	X =  480.566  mm,	Y =   -445.856  mm,	Z =   -229.363  mm,
	W =  90.000 deg,	P =   0.000 deg,	R =   90.000 deg
};
P[2287]{
   GP1:
	UF : 0, UT : 6,		CONFIG : 'N U T, 0, 0, 0',
	X =  481.182  mm,	Y =   -445.586  mm,	Z =   -229.154  mm,
	W =  90.000 deg,	P =   0.000 deg,	R =   90.000 deg
};
P[2288]{
   GP1:
	UF : 0, UT : 6,		CONFIG : 'N U T, 0, 0, 0',
	X =  482.170  mm,	Y =   -444.919  mm,	Z =   -229.387  mm,
	W =  90.000 deg,	P =   0.000 deg,	R =   90.000 deg
};
P[2289]{
   GP1:
	UF : 0, UT : 6,		CONFIG : 'N U T, 0, 0, 0',
	X =  483.233  mm,	Y =   -444.478  mm,	Z =   -228.968  mm,
	W =  90.000 deg,	P =   0.000 deg,	R =   90.000 deg
};
P[2290]{
   GP1:
	UF : 0, UT : 6,		CONFIG : 'N U T, 0, 0, 0',
	X =  484.850  mm,	Y =   -443.422  mm,	Z =   -229.266  mm,
	W =  90.000 deg,	P =   0.000 deg,	R =   90.000 deg
};
P[2291]{
   GP1:
	UF : 0, UT : 6,		CONFIG : 'N U T, 0, 0, 0',
	X =  485.668  mm,	Y =   -442.930  mm,	Z =   -229.313  mm,
	W =  90.000 deg,	P =   0.000 deg,	R =   90.000 deg
};
P[2292]{
   GP1:
	UF : 0, UT : 6,		CONFIG : 'N U T, 0, 0, 0',
	X =  487.431  mm,	Y =   -441.948  mm,	Z =   -229.227  mm,
	W =  90.000 deg,	P =   0.000 deg,	R =   90.000 deg
};
P[2293]{
   GP1:
	UF : 0, UT : 6,		CONFIG : 'N U T, 0, 0, 0',
	X =  488.798  mm,	Y =   -441.282  mm,	Z =   -228.926  mm,
	W =  90.000 deg,	P =   0.000 deg,	R =   90.000 deg
};
P[2294]{
   GP1:
	UF : 0, UT : 6,		CONFIG : 'N U T, 0, 0, 0',
	X =  492.018  mm,	Y =   -439.329  mm,	Z =   -229.155  mm,
	W =  90.000 deg,	P =   0.000 deg,	R =   90.000 deg
};
P[2295]{
   GP1:
	UF : 0, UT : 6,		CONFIG : 'N U T, 0, 0, 0',
	X =  493.252  mm,	Y =   -438.538  mm,	Z =   -229.345  mm,
	W =  90.000 deg,	P =   0.000 deg,	R =   90.000 deg
};
P[2296]{
   GP1:
	UF : 0, UT : 6,		CONFIG : 'N U T, 0, 0, 0',
	X =  494.374  mm,	Y =   -438.005  mm,	Z =   -229.066  mm,
	W =  90.000 deg,	P =   0.000 deg,	R =   90.000 deg
};
P[2297]{
   GP1:
	UF : 0, UT : 6,		CONFIG : 'N U T, 0, 0, 0',
	X =  495.502  mm,	Y =   -437.305  mm,	Z =   -229.186  mm,
	W =  90.000 deg,	P =   0.000 deg,	R =   90.000 deg
};
P[2298]{
   GP1:
	UF : 0, UT : 6,		CONFIG : 'N U T, 0, 0, 0',
	X =  496.386  mm,	Y =   -436.731  mm,	Z =   -229.340  mm,
	W =  90.000 deg,	P =   0.000 deg,	R =   90.000 deg
};
P[2299]{
   GP1:
	UF : 0, UT : 6,		CONFIG : 'N U T, 0, 0, 0',
	X =  497.271  mm,	Y =   -436.217  mm,	Z =   -229.347  mm,
	W =  90.000 deg,	P =   0.000 deg,	R =   90.000 deg
};
P[2300]{
   GP1:
	UF : 0, UT : 6,		CONFIG : 'N U T, 0, 0, 0',
	X =  498.310  mm,	Y =   -435.633  mm,	Z =   -229.309  mm,
	W =  90.000 deg,	P =   0.000 deg,	R =   90.000 deg
};
P[2301]{
   GP1:
	UF : 0, UT : 6,		CONFIG : 'N U T, 0, 0, 0',
	X =  499.714  mm,	Y =   -434.837  mm,	Z =   -229.273  mm,
	W =  90.000 deg,	P =   0.000 deg,	R =   90.000 deg
};
P[2302]{
   GP1:
	UF : 0, UT : 6,		CONFIG : 'N U T, 0, 0, 0',
	X =  500.828  mm,	Y =   -434.198  mm,	Z =   -229.203  mm,
	W =  90.000 deg,	P =   0.000 deg,	R =   90.000 deg
};
P[2303]{
   GP1:
	UF : 0, UT : 6,		CONFIG : 'N U T, 0, 0, 0',
	X =  502.097  mm,	Y =   -433.246  mm,	Z =   -229.316  mm,
	W =  90.000 deg,	P =   0.000 deg,	R =   90.000 deg
};
P[2304]{
   GP1:
	UF : 0, UT : 6,		CONFIG : 'N U T, 0, 0, 0',
	X =  503.730  mm,	Y =   -431.797  mm,	Z =   -229.261  mm,
	W =  90.000 deg,	P =   0.000 deg,	R =   90.000 deg
};
P[2305]{
   GP1:
	UF : 0, UT : 6,		CONFIG : 'N U T, 0, 0, 0',
	X =  504.332  mm,	Y =   -431.117  mm,	Z =   -229.304  mm,
	W =  90.000 deg,	P =   0.000 deg,	R =   90.000 deg
};
P[2306]{
   GP1:
	UF : 0, UT : 6,		CONFIG : 'N U T, 0, 0, 0',
	X =  505.528  mm,	Y =   -429.350  mm,	Z =   -229.315  mm,
	W =  90.000 deg,	P =   0.000 deg,	R =   90.000 deg
};
P[2307]{
   GP1:
	UF : 0, UT : 6,		CONFIG : 'N U T, 0, 0, 0',
	X =  506.145  mm,	Y =   -428.643  mm,	Z =   -228.908  mm,
	W =  90.000 deg,	P =   0.000 deg,	R =   90.000 deg
};
P[2308]{
   GP1:
	UF : 0, UT : 6,		CONFIG : 'N U T, 0, 0, 0',
	X =  506.322  mm,	Y =   -427.681  mm,	Z =   -229.271  mm,
	W =  90.000 deg,	P =   0.000 deg,	R =   90.000 deg
};
P[2309]{
   GP1:
	UF : 0, UT : 6,		CONFIG : 'N U T, 0, 0, 0',
	X =  506.669  mm,	Y =   -427.189  mm,	Z =   -228.972  mm,
	W =  90.000 deg,	P =   0.000 deg,	R =   90.000 deg
};
P[2310]{
   GP1:
	UF : 0, UT : 6,		CONFIG : 'N U T, 0, 0, 0',
	X =  507.163  mm,	Y =   -425.222  mm,	Z =   -228.904  mm,
	W =  90.000 deg,	P =   0.000 deg,	R =   90.000 deg
};
P[2311]{
   GP1:
	UF : 0, UT : 6,		CONFIG : 'N U T, 0, 0, 0',
	X =  507.195  mm,	Y =   -423.814  mm,	Z =   -229.152  mm,
	W =  90.000 deg,	P =   0.000 deg,	R =   90.000 deg
};
P[2312]{
   GP1:
	UF : 0, UT : 6,		CONFIG : 'N U T, 0, 0, 0',
	X =  506.821  mm,	Y =   -419.984  mm,	Z =   -228.966  mm,
	W =  90.000 deg,	P =   0.000 deg,	R =   90.000 deg
};
P[2313]{
   GP1:
	UF : 0, UT : 6,		CONFIG : 'N U T, 0, 0, 0',
	X =  506.580  mm,	Y =   -419.034  mm,	Z =   -228.929  mm,
	W =  90.000 deg,	P =   0.000 deg,	R =   90.000 deg
};
P[2314]{
   GP1:
	UF : 0, UT : 6,		CONFIG : 'N U T, 0, 0, 0',
	X =  506.090  mm,	Y =   -418.254  mm,	Z =   -229.258  mm,
	W =  90.000 deg,	P =   0.000 deg,	R =   90.000 deg
};
P[2315]{
   GP1:
	UF : 0, UT : 6,		CONFIG : 'N U T, 0, 0, 0',
	X =  505.684  mm,	Y =   -417.150  mm,	Z =   -229.023  mm,
	W =  90.000 deg,	P =   0.000 deg,	R =   90.000 deg
};
P[2316]{
   GP1:
	UF : 0, UT : 6,		CONFIG : 'N U T, 0, 0, 0',
	X =  505.249  mm,	Y =   -416.523  mm,	Z =   -229.335  mm,
	W =  90.000 deg,	P =   0.000 deg,	R =   90.000 deg
};
P[2317]{
   GP1:
	UF : 0, UT : 6,		CONFIG : 'N U T, 0, 0, 0',
	X =  504.966  mm,	Y =   -415.874  mm,	Z =   -229.110  mm,
	W =  90.000 deg,	P =   0.000 deg,	R =   90.000 deg
};
P[2318]{
   GP1:
	UF : 0, UT : 6,		CONFIG : 'N U T, 0, 0, 0',
	X =  504.322  mm,	Y =   -414.678  mm,	Z =   -228.999  mm,
	W =  90.000 deg,	P =   0.000 deg,	R =   90.000 deg
};
P[2319]{
   GP1:
	UF : 0, UT : 6,		CONFIG : 'N U T, 0, 0, 0',
	X =  501.872  mm,	Y =   -410.680  mm,	Z =   -229.341  mm,
	W =  90.000 deg,	P =   0.000 deg,	R =   90.000 deg
};
P[2320]{
   GP1:
	UF : 0, UT : 6,		CONFIG : 'N U T, 0, 0, 0',
	X =  501.465  mm,	Y =   -409.684  mm,	Z =   -228.933  mm,
	W =  90.000 deg,	P =   0.000 deg,	R =   90.000 deg
};
P[2321]{
   GP1:
	UF : 0, UT : 6,		CONFIG : 'N U T, 0, 0, 0',
	X =  500.200  mm,	Y =   -407.765  mm,	Z =   -229.313  mm,
	W =  90.000 deg,	P =   0.000 deg,	R =   90.000 deg
};
P[2322]{
   GP1:
	UF : 0, UT : 6,		CONFIG : 'N U T, 0, 0, 0',
	X =  499.334  mm,	Y =   -406.182  mm,	Z =   -229.197  mm,
	W =  90.000 deg,	P =   0.000 deg,	R =   90.000 deg
};
P[2323]{
   GP1:
	UF : 0, UT : 6,		CONFIG : 'N U T, 0, 0, 0',
	X =  496.746  mm,	Y =   -401.722  mm,	Z =   -229.228  mm,
	W =  90.000 deg,	P =   0.000 deg,	R =   90.000 deg
};
P[2324]{
   GP1:
	UF : 0, UT : 6,		CONFIG : 'N U T, 0, 0, 0',
	X =  495.091  mm,	Y =   -398.847  mm,	Z =   -229.216  mm,
	W =  90.000 deg,	P =   0.000 deg,	R =   90.000 deg
};
P[2325]{
   GP1:
	UF : 0, UT : 6,		CONFIG : 'N U T, 0, 0, 0',
	X =  493.661  mm,	Y =   -396.466  mm,	Z =   -229.351  mm,
	W =  90.000 deg,	P =   0.000 deg,	R =   90.000 deg
};
P[2326]{
   GP1:
	UF : 0, UT : 6,		CONFIG : 'N U T, 0, 0, 0',
	X =  491.412  mm,	Y =   -392.372  mm,	Z =   -229.073  mm,
	W =  90.000 deg,	P =   0.000 deg,	R =   90.000 deg
};
P[2327]{
   GP1:
	UF : 0, UT : 6,		CONFIG : 'N U T, 0, 0, 0',
	X =  490.971  mm,	Y =   -391.504  mm,	Z =   -228.926  mm,
	W =  90.000 deg,	P =   0.000 deg,	R =   90.000 deg
};
P[2328]{
   GP1:
	UF : 0, UT : 6,		CONFIG : 'N U T, 0, 0, 0',
	X =  490.552  mm,	Y =   -390.879  mm,	Z =   -229.066  mm,
	W =  90.000 deg,	P =   0.000 deg,	R =   90.000 deg
};
P[2329]{
   GP1:
	UF : 0, UT : 6,		CONFIG : 'N U T, 0, 0, 0',
	X =  489.653  mm,	Y =   -389.328  mm,	Z =   -229.076  mm,
	W =  90.000 deg,	P =   0.000 deg,	R =   90.000 deg
};
P[2330]{
   GP1:
	UF : 0, UT : 6,		CONFIG : 'N U T, 0, 0, 0',
	X =  488.589  mm,	Y =   -387.690  mm,	Z =   -229.362  mm,
	W =  90.000 deg,	P =   0.000 deg,	R =   90.000 deg
};
P[2331]{
   GP1:
	UF : 0, UT : 6,		CONFIG : 'N U T, 0, 0, 0',
	X =  487.058  mm,	Y =   -385.020  mm,	Z =   -229.336  mm,
	W =  90.000 deg,	P =   0.000 deg,	R =   90.000 deg
};
P[2332]{
   GP1:
	UF : 0, UT : 6,		CONFIG : 'N U T, 0, 0, 0',
	X =  486.583  mm,	Y =   -383.988  mm,	Z =   -229.041  mm,
	W =  90.000 deg,	P =   0.000 deg,	R =   90.000 deg
};
P[2333]{
   GP1:
	UF : 0, UT : 6,		CONFIG : 'N U T, 0, 0, 0',
	X =  485.210  mm,	Y =   -381.630  mm,	Z =   -229.073  mm,
	W =  90.000 deg,	P =   0.000 deg,	R =   90.000 deg
};
P[2334]{
   GP1:
	UF : 0, UT : 6,		CONFIG : 'N U T, 0, 0, 0',
	X =  484.643  mm,	Y =   -380.536  mm,	Z =   -228.913  mm,
	W =  90.000 deg,	P =   0.000 deg,	R =   90.000 deg
};
P[2335]{
   GP1:
	UF : 0, UT : 6,		CONFIG : 'N U T, 0, 0, 0',
	X =  483.687  mm,	Y =   -379.150  mm,	Z =   -229.294  mm,
	W =  90.000 deg,	P =   0.000 deg,	R =   90.000 deg
};
P[2336]{
   GP1:
	UF : 0, UT : 6,		CONFIG : 'N U T, 0, 0, 0',
	X =  482.653  mm,	Y =   -377.218  mm,	Z =   -229.093  mm,
	W =  90.000 deg,	P =   0.000 deg,	R =   90.000 deg
};
P[2337]{
   GP1:
	UF : 0, UT : 6,		CONFIG : 'N U T, 0, 0, 0',
	X =  482.012  mm,	Y =   -376.031  mm,	Z =   -228.986  mm,
	W =  90.000 deg,	P =   0.000 deg,	R =   90.000 deg
};
P[2338]{
   GP1:
	UF : 0, UT : 6,		CONFIG : 'N U T, 0, 0, 0',
	X =  481.638  mm,	Y =   -375.643  mm,	Z =   -229.351  mm,
	W =  90.000 deg,	P =   0.000 deg,	R =   90.000 deg
};
P[2339]{
   GP1:
	UF : 0, UT : 6,		CONFIG : 'N U T, 0, 0, 0',
	X =  480.478  mm,	Y =   -373.530  mm,	Z =   -229.204  mm,
	W =  90.000 deg,	P =   0.000 deg,	R =   90.000 deg
};
P[2340]{
   GP1:
	UF : 0, UT : 6,		CONFIG : 'N U T, 0, 0, 0',
	X =  478.950  mm,	Y =   -371.001  mm,	Z =   -229.370  mm,
	W =  90.000 deg,	P =   0.000 deg,	R =   90.000 deg
};
P[2341]{
   GP1:
	UF : 0, UT : 6,		CONFIG : 'N U T, 0, 0, 0',
	X =  478.603  mm,	Y =   -370.100  mm,	Z =   -228.948  mm,
	W =  90.000 deg,	P =   0.000 deg,	R =   90.000 deg
};
P[2342]{
   GP1:
	UF : 0, UT : 6,		CONFIG : 'N U T, 0, 0, 0',
	X =  478.005  mm,	Y =   -369.237  mm,	Z =   -229.192  mm,
	W =  90.000 deg,	P =   0.000 deg,	R =   90.000 deg
};
P[2343]{
   GP1:
	UF : 0, UT : 6,		CONFIG : 'N U T, 0, 0, 0',
	X =  476.529  mm,	Y =   -366.505  mm,	Z =   -228.945  mm,
	W =  90.000 deg,	P =   0.000 deg,	R =   90.000 deg
};
P[2344]{
   GP1:
	UF : 0, UT : 6,		CONFIG : 'N U T, 0, 0, 0',
	X =  475.840  mm,	Y =   -365.565  mm,	Z =   -229.297  mm,
	W =  90.000 deg,	P =   0.000 deg,	R =   90.000 deg
};
P[2345]{
   GP1:
	UF : 0, UT : 6,		CONFIG : 'N U T, 0, 0, 0',
	X =  475.226  mm,	Y =   -364.521  mm,	Z =   -229.327  mm,
	W =  90.000 deg,	P =   0.000 deg,	R =   90.000 deg
};
P[2346]{
   GP1:
	UF : 0, UT : 6,		CONFIG : 'N U T, 0, 0, 0',
	X =  474.947  mm,	Y =   -363.892  mm,	Z =   -229.122  mm,
	W =  90.000 deg,	P =   0.000 deg,	R =   90.000 deg
};
P[2347]{
   GP1:
	UF : 0, UT : 6,		CONFIG : 'N U T, 0, 0, 0',
	X =  474.268  mm,	Y =   -362.568  mm,	Z =   -228.915  mm,
	W =  90.000 deg,	P =   0.000 deg,	R =   90.000 deg
};
P[2348]{
   GP1:
	UF : 0, UT : 6,		CONFIG : 'N U T, 0, 0, 0',
	X =  473.577  mm,	Y =   -361.591  mm,	Z =   -229.222  mm,
	W =  90.000 deg,	P =   0.000 deg,	R =   90.000 deg
};
P[2349]{
   GP1:
	UF : 0, UT : 6,		CONFIG : 'N U T, 0, 0, 0',
	X =  472.899  mm,	Y =   -360.264  mm,	Z =   -229.008  mm,
	W =  90.000 deg,	P =   0.000 deg,	R =   90.000 deg
};
P[2350]{
   GP1:
	UF : 0, UT : 6,		CONFIG : 'N U T, 0, 0, 0',
	X =  471.935  mm,	Y =   -358.624  mm,	Z =   -229.049  mm,
	W =  90.000 deg,	P =   0.000 deg,	R =   90.000 deg
};
P[2351]{
   GP1:
	UF : 0, UT : 6,		CONFIG : 'N U T, 0, 0, 0',
	X =  471.530  mm,	Y =   -358.012  mm,	Z =   -229.175  mm,
	W =  90.000 deg,	P =   0.000 deg,	R =   90.000 deg
};
P[2352]{
   GP1:
	UF : 0, UT : 6,		CONFIG : 'N U T, 0, 0, 0',
	X =  470.504  mm,	Y =   -356.359  mm,	Z =   -229.350  mm,
	W =  90.000 deg,	P =   0.000 deg,	R =   90.000 deg
};
P[2353]{
   GP1:
	UF : 0, UT : 6,		CONFIG : 'N U T, 0, 0, 0',
	X =  469.943  mm,	Y =   -355.369  mm,	Z =   -229.324  mm,
	W =  90.000 deg,	P =   0.000 deg,	R =   90.000 deg
};
P[2354]{
   GP1:
	UF : 0, UT : 6,		CONFIG : 'N U T, 0, 0, 0',
	X =  469.352  mm,	Y =   -354.235  mm,	Z =   -229.169  mm,
	W =  90.000 deg,	P =   0.000 deg,	R =   90.000 deg
};
P[2355]{
   GP1:
	UF : 0, UT : 6,		CONFIG : 'N U T, 0, 0, 0',
	X =  467.793  mm,	Y =   -351.354  mm,	Z =   -228.914  mm,
	W =  90.000 deg,	P =   0.000 deg,	R =   90.000 deg
};
P[2356]{
   GP1:
	UF : 0, UT : 6,		CONFIG : 'N U T, 0, 0, 0',
	X =  467.124  mm,	Y =   -350.435  mm,	Z =   -229.252  mm,
	W =  90.000 deg,	P =   0.000 deg,	R =   90.000 deg
};
P[2357]{
   GP1:
	UF : 0, UT : 6,		CONFIG : 'N U T, 0, 0, 0',
	X =  466.834  mm,	Y =   -349.690  mm,	Z =   -228.910  mm,
	W =  90.000 deg,	P =   0.000 deg,	R =   90.000 deg
};
P[2358]{
   GP1:
	UF : 0, UT : 6,		CONFIG : 'N U T, 0, 0, 0',
	X =  465.959  mm,	Y =   -348.178  mm,	Z =   -228.914  mm,
	W =  90.000 deg,	P =   0.000 deg,	R =   90.000 deg
};
P[2359]{
   GP1:
	UF : 0, UT : 6,		CONFIG : 'N U T, 0, 0, 0',
	X =  465.404  mm,	Y =   -347.437  mm,	Z =   -229.227  mm,
	W =  90.000 deg,	P =   0.000 deg,	R =   90.000 deg
};
P[2360]{
   GP1:
	UF : 0, UT : 6,		CONFIG : 'N U T, 0, 0, 0',
	X =  464.736  mm,	Y =   -346.319  mm,	Z =   -229.280  mm,
	W =  90.000 deg,	P =   0.000 deg,	R =   90.000 deg
};
P[2361]{
   GP1:
	UF : 0, UT : 6,		CONFIG : 'N U T, 0, 0, 0',
	X =  464.332  mm,	Y =   -345.434  mm,	Z =   -229.017  mm,
	W =  90.000 deg,	P =   0.000 deg,	R =   90.000 deg
};
P[2362]{
   GP1:
	UF : 0, UT : 6,		CONFIG : 'N U T, 0, 0, 0',
	X =  463.800  mm,	Y =   -344.455  mm,	Z =   -228.940  mm,
	W =  90.000 deg,	P =   0.000 deg,	R =   90.000 deg
};
P[2363]{
   GP1:
	UF : 0, UT : 6,		CONFIG : 'N U T, 0, 0, 0',
	X =  463.406  mm,	Y =   -344.003  mm,	Z =   -229.262  mm,
	W =  90.000 deg,	P =   0.000 deg,	R =   90.000 deg
};
P[2364]{
   GP1:
	UF : 0, UT : 6,		CONFIG : 'N U T, 0, 0, 0',
	X =  463.015  mm,	Y =   -343.412  mm,	Z =   -229.383  mm,
	W =  90.000 deg,	P =   0.000 deg,	R =   90.000 deg
};
P[2365]{
   GP1:
	UF : 0, UT : 6,		CONFIG : 'N U T, 0, 0, 0',
	X =  462.606  mm,	Y =   -342.592  mm,	Z =   -229.228  mm,
	W =  90.000 deg,	P =   0.000 deg,	R =   90.000 deg
};
P[2366]{
   GP1:
	UF : 0, UT : 6,		CONFIG : 'N U T, 0, 0, 0',
	X =  461.923  mm,	Y =   -341.496  mm,	Z =   -229.350  mm,
	W =  90.000 deg,	P =   0.000 deg,	R =   90.000 deg
};
P[2367]{
   GP1:
	UF : 0, UT : 6,		CONFIG : 'N U T, 0, 0, 0',
	X =  461.418  mm,	Y =   -340.391  mm,	Z =   -229.027  mm,
	W =  90.000 deg,	P =   0.000 deg,	R =   90.000 deg
};
P[2368]{
   GP1:
	UF : 0, UT : 6,		CONFIG : 'N U T, 0, 0, 0',
	X =  461.027  mm,	Y =   -339.939  mm,	Z =   -229.343  mm,
	W =  90.000 deg,	P =   0.000 deg,	R =   90.000 deg
};
P[2369]{
   GP1:
	UF : 0, UT : 6,		CONFIG : 'N U T, 0, 0, 0',
	X =  460.237  mm,	Y =   -338.429  mm,	Z =   -229.141  mm,
	W =  90.000 deg,	P =   0.000 deg,	R =   90.000 deg
};
P[2370]{
   GP1:
	UF : 0, UT : 6,		CONFIG : 'N U T, 0, 0, 0',
	X =  459.232  mm,	Y =   -336.565  mm,	Z =   -228.969  mm,
	W =  90.000 deg,	P =   0.000 deg,	R =   90.000 deg
};
P[2371]{
   GP1:
	UF : 0, UT : 6,		CONFIG : 'N U T, 0, 0, 0',
	X =  458.669  mm,	Y =   -335.549  mm,	Z =   -228.911  mm,
	W =  90.000 deg,	P =   0.000 deg,	R =   90.000 deg
};
P[2372]{
   GP1:
	UF : 0, UT : 6,		CONFIG : 'N U T, 0, 0, 0',
	X =  458.273  mm,	Y =   -335.200  mm,	Z =   -229.384  mm,
	W =  90.000 deg,	P =   0.000 deg,	R =   90.000 deg
};
P[2373]{
   GP1:
	UF : 0, UT : 6,		CONFIG : 'N U T, 0, 0, 0',
	X =  456.601  mm,	Y =   -331.959  mm,	Z =   -228.900  mm,
	W =  90.000 deg,	P =   0.000 deg,	R =   90.000 deg
};
P[2374]{
   GP1:
	UF : 0, UT : 6,		CONFIG : 'N U T, 0, 0, 0',
	X =  456.178  mm,	Y =   -331.310  mm,	Z =   -229.018  mm,
	W =  90.000 deg,	P =   0.000 deg,	R =   90.000 deg
};
P[2375]{
   GP1:
	UF : 0, UT : 6,		CONFIG : 'N U T, 0, 0, 0',
	X =  455.776  mm,	Y =   -330.629  mm,	Z =   -229.039  mm,
	W =  90.000 deg,	P =   0.000 deg,	R =   90.000 deg
};
P[2376]{
   GP1:
	UF : 0, UT : 6,		CONFIG : 'N U T, 0, 0, 0',
	X =  454.651  mm,	Y =   -328.902  mm,	Z =   -229.349  mm,
	W =  90.000 deg,	P =   0.000 deg,	R =   90.000 deg
};
P[2377]{
   GP1:
	UF : 0, UT : 6,		CONFIG : 'N U T, 0, 0, 0',
	X =  453.814  mm,	Y =   -327.302  mm,	Z =   -229.140  mm,
	W =  90.000 deg,	P =   0.000 deg,	R =   90.000 deg
};
P[2378]{
   GP1:
	UF : 0, UT : 6,		CONFIG : 'N U T, 0, 0, 0',
	X =  453.457  mm,	Y =   -326.686  mm,	Z =   -229.141  mm,
	W =  90.000 deg,	P =   0.000 deg,	R =   90.000 deg
};
P[2379]{
   GP1:
	UF : 0, UT : 6,		CONFIG : 'N U T, 0, 0, 0',
	X =  453.136  mm,	Y =   -326.062  mm,	Z =   -229.047  mm,
	W =  90.000 deg,	P =   0.000 deg,	R =   90.000 deg
};
P[2380]{
   GP1:
	UF : 0, UT : 6,		CONFIG : 'N U T, 0, 0, 0',
	X =  451.971  mm,	Y =   -324.078  mm,	Z =   -229.094  mm,
	W =  90.000 deg,	P =   0.000 deg,	R =   90.000 deg
};
P[2381]{
   GP1:
	UF : 0, UT : 6,		CONFIG : 'N U T, 0, 0, 0',
	X =  449.559  mm,	Y =   -319.786  mm,	Z =   -228.935  mm,
	W =  90.000 deg,	P =   0.000 deg,	R =   90.000 deg
};
P[2382]{
   GP1:
	UF : 0, UT : 6,		CONFIG : 'N U T, 0, 0, 0',
	X =  448.790  mm,	Y =   -318.576  mm,	Z =   -229.103  mm,
	W =  90.000 deg,	P =   0.000 deg,	R =   90.000 deg
};
P[2383]{
   GP1:
	UF : 0, UT : 6,		CONFIG : 'N U T, 0, 0, 0',
	X =  446.954  mm,	Y =   -315.552  mm,	Z =   -229.321  mm,
	W =  90.000 deg,	P =   0.000 deg,	R =   90.000 deg
};
P[2384]{
   GP1:
	UF : 0, UT : 6,		CONFIG : 'N U T, 0, 0, 0',
	X =  446.659  mm,	Y =   -314.936  mm,	Z =   -229.175  mm,
	W =  90.000 deg,	P =   0.000 deg,	R =   90.000 deg
};
P[2385]{
   GP1:
	UF : 0, UT : 6,		CONFIG : 'N U T, 0, 0, 0',
	X =  446.120  mm,	Y =   -314.042  mm,	Z =   -229.229  mm,
	W =  90.000 deg,	P =   0.000 deg,	R =   90.000 deg
};
P[2386]{
   GP1:
	UF : 0, UT : 6,		CONFIG : 'N U T, 0, 0, 0',
	X =  444.698  mm,	Y =   -311.514  mm,	Z =   -229.140  mm,
	W =  90.000 deg,	P =   0.000 deg,	R =   90.000 deg
};
P[2387]{
   GP1:
	UF : 0, UT : 6,		CONFIG : 'N U T, 0, 0, 0',
	X =  444.342  mm,	Y =   -310.953  mm,	Z =   -229.216  mm,
	W =  90.000 deg,	P =   0.000 deg,	R =   90.000 deg
};
P[2388]{
   GP1:
	UF : 0, UT : 6,		CONFIG : 'N U T, 0, 0, 0',
	X =  444.092  mm,	Y =   -310.296  mm,	Z =   -228.903  mm,
	W =  90.000 deg,	P =   0.000 deg,	R =   90.000 deg
};
P[2389]{
   GP1:
	UF : 0, UT : 6,		CONFIG : 'N U T, 0, 0, 0',
	X =  442.535  mm,	Y =   -307.939  mm,	Z =   -229.379  mm,
	W =  90.000 deg,	P =   0.000 deg,	R =   90.000 deg
};
P[2390]{
   GP1:
	UF : 0, UT : 6,		CONFIG : 'N U T, 0, 0, 0',
	X =  440.875  mm,	Y =   -304.766  mm,	Z =   -228.958  mm,
	W =  90.000 deg,	P =   0.000 deg,	R =   90.000 deg
};
P[2391]{
   GP1:
	UF : 0, UT : 6,		CONFIG : 'N U T, 0, 0, 0',
	X =  440.370  mm,	Y =   -303.954  mm,	Z =   -229.051  mm,
	W =  90.000 deg,	P =   0.000 deg,	R =   90.000 deg
};
P[2392]{
   GP1:
	UF : 0, UT : 6,		CONFIG : 'N U T, 0, 0, 0',
	X =  439.191  mm,	Y =   -302.015  mm,	Z =   -229.194  mm,
	W =  90.000 deg,	P =   0.000 deg,	R =   90.000 deg
};
P[2393]{
   GP1:
	UF : 0, UT : 6,		CONFIG : 'N U T, 0, 0, 0',
	X =  438.809  mm,	Y =   -301.361  mm,	Z =   -229.205  mm,
	W =  90.000 deg,	P =   0.000 deg,	R =   90.000 deg
};
P[2394]{
   GP1:
	UF : 0, UT : 6,		CONFIG : 'N U T, 0, 0, 0',
	X =  438.201  mm,	Y =   -300.439  mm,	Z =   -229.387  mm,
	W =  90.000 deg,	P =   0.000 deg,	R =   90.000 deg
};
P[2395]{
   GP1:
	UF : 0, UT : 6,		CONFIG : 'N U T, 0, 0, 0',
	X =  436.533  mm,	Y =   -297.317  mm,	Z =   -229.061  mm,
	W =  90.000 deg,	P =   0.000 deg,	R =   90.000 deg
};
P[2396]{
   GP1:
	UF : 0, UT : 6,		CONFIG : 'N U T, 0, 0, 0',
	X =  435.638  mm,	Y =   -295.709  mm,	Z =   -228.979  mm,
	W =  90.000 deg,	P =   0.000 deg,	R =   90.000 deg
};
P[2397]{
   GP1:
	UF : 0, UT : 6,		CONFIG : 'N U T, 0, 0, 0',
	X =  434.295  mm,	Y =   -293.622  mm,	Z =   -229.313  mm,
	W =  90.000 deg,	P =   0.000 deg,	R =   90.000 deg
};
P[2398]{
   GP1:
	UF : 0, UT : 6,		CONFIG : 'N U T, 0, 0, 0',
	X =  433.936  mm,	Y =   -292.975  mm,	Z =   -229.278  mm,
	W =  90.000 deg,	P =   0.000 deg,	R =   90.000 deg
};
P[2399]{
   GP1:
	UF : 0, UT : 6,		CONFIG : 'N U T, 0, 0, 0',
	X =  433.468  mm,	Y =   -292.209  mm,	Z =   -229.341  mm,
	W =  90.000 deg,	P =   0.000 deg,	R =   90.000 deg
};
P[2400]{
   GP1:
	UF : 0, UT : 6,		CONFIG : 'N U T, 0, 0, 0',
	X =  430.840  mm,	Y =   -287.594  mm,	Z =   -229.251  mm,
	W =  90.000 deg,	P =   0.000 deg,	R =   90.000 deg
};
P[2401]{
   GP1:
	UF : 0, UT : 6,		CONFIG : 'N U T, 0, 0, 0',
	X =  430.476  mm,	Y =   -286.901  mm,	Z =   -229.166  mm,
	W =  90.000 deg,	P =   0.000 deg,	R =   90.000 deg
};
P[2402]{
   GP1:
	UF : 0, UT : 6,		CONFIG : 'N U T, 0, 0, 0',
	X =  429.790  mm,	Y =   -285.601  mm,	Z =   -229.009  mm,
	W =  90.000 deg,	P =   0.000 deg,	R =   90.000 deg
};
P[2403]{
   GP1:
	UF : 0, UT : 6,		CONFIG : 'N U T, 0, 0, 0',
	X =  429.351  mm,	Y =   -285.097  mm,	Z =   -229.368  mm,
	W =  90.000 deg,	P =   0.000 deg,	R =   90.000 deg
};
P[2404]{
   GP1:
	UF : 0, UT : 6,		CONFIG : 'N U T, 0, 0, 0',
	X =  428.977  mm,	Y =   -284.223  mm,	Z =   -229.050  mm,
	W =  90.000 deg,	P =   0.000 deg,	R =   90.000 deg
};
P[2405]{
   GP1:
	UF : 0, UT : 6,		CONFIG : 'N U T, 0, 0, 0',
	X =  428.460  mm,	Y =   -283.449  mm,	Z =   -229.219  mm,
	W =  90.000 deg,	P =   0.000 deg,	R =   90.000 deg
};
P[2406]{
   GP1:
	UF : 0, UT : 6,		CONFIG : 'N U T, 0, 0, 0',
	X =  426.700  mm,	Y =   -280.198  mm,	Z =   -228.936  mm,
	W =  90.000 deg,	P =   0.000 deg,	R =   90.000 deg
};
P[2407]{
   GP1:
	UF : 0, UT : 6,		CONFIG : 'N U T, 0, 0, 0',
	X =  425.962  mm,	Y =   -278.911  mm,	Z =   -228.924  mm,
	W =  90.000 deg,	P =   0.000 deg,	R =   90.000 deg
};
P[2408]{
   GP1:
	UF : 0, UT : 6,		CONFIG : 'N U T, 0, 0, 0',
	X =  424.302  mm,	Y =   -276.072  mm,	Z =   -228.971  mm,
	W =  90.000 deg,	P =   0.000 deg,	R =   90.000 deg
};
P[2409]{
   GP1:
	UF : 0, UT : 6,		CONFIG : 'N U T, 0, 0, 0',
	X =  422.750  mm,	Y =   -273.408  mm,	Z =   -229.010  mm,
	W =  90.000 deg,	P =   0.000 deg,	R =   90.000 deg
};
P[2410]{
   GP1:
	UF : 0, UT : 6,		CONFIG : 'N U T, 0, 0, 0',
	X =  422.369  mm,	Y =   -272.752  mm,	Z =   -229.014  mm,
	W =  90.000 deg,	P =   0.000 deg,	R =   90.000 deg
};
P[2411]{
   GP1:
	UF : 0, UT : 6,		CONFIG : 'N U T, 0, 0, 0',
	X =  421.027  mm,	Y =   -270.684  mm,	Z =   -229.372  mm,
	W =  90.000 deg,	P =   0.000 deg,	R =   90.000 deg
};
P[2412]{
   GP1:
	UF : 0, UT : 6,		CONFIG : 'N U T, 0, 0, 0',
	X =  420.123  mm,	Y =   -268.967  mm,	Z =   -229.160  mm,
	W =  90.000 deg,	P =   0.000 deg,	R =   90.000 deg
};
P[2413]{
   GP1:
	UF : 0, UT : 6,		CONFIG : 'N U T, 0, 0, 0',
	X =  419.772  mm,	Y =   -268.392  mm,	Z =   -229.207  mm,
	W =  90.000 deg,	P =   0.000 deg,	R =   90.000 deg
};
P[2414]{
   GP1:
	UF : 0, UT : 6,		CONFIG : 'N U T, 0, 0, 0',
	X =  419.099  mm,	Y =   -267.146  mm,	Z =   -229.093  mm,
	W =  90.000 deg,	P =   0.000 deg,	R =   90.000 deg
};
P[2415]{
   GP1:
	UF : 0, UT : 6,		CONFIG : 'N U T, 0, 0, 0',
	X =  417.965  mm,	Y =   -265.231  mm,	Z =   -229.162  mm,
	W =  90.000 deg,	P =   0.000 deg,	R =   90.000 deg
};
P[2416]{
   GP1:
	UF : 0, UT : 6,		CONFIG : 'N U T, 0, 0, 0',
	X =  417.150  mm,	Y =   -263.903  mm,	Z =   -229.279  mm,
	W =  90.000 deg,	P =   0.000 deg,	R =   90.000 deg
};
P[2417]{
   GP1:
	UF : 0, UT : 6,		CONFIG : 'N U T, 0, 0, 0',
	X =  415.506  mm,	Y =   -260.954  mm,	Z =   -229.137  mm,
	W =  90.000 deg,	P =   0.000 deg,	R =   90.000 deg
};
P[2418]{
   GP1:
	UF : 0, UT : 6,		CONFIG : 'N U T, 0, 0, 0',
	X =  414.446  mm,	Y =   -259.189  mm,	Z =   -229.235  mm,
	W =  90.000 deg,	P =   0.000 deg,	R =   90.000 deg
};
P[2419]{
   GP1:
	UF : 0, UT : 6,		CONFIG : 'N U T, 0, 0, 0',
	X =  413.559  mm,	Y =   -257.419  mm,	Z =   -228.908  mm,
	W =  90.000 deg,	P =   0.000 deg,	R =   90.000 deg
};
P[2420]{
   GP1:
	UF : 0, UT : 6,		CONFIG : 'N U T, 0, 0, 0',
	X =  412.900  mm,	Y =   -256.470  mm,	Z =   -229.177  mm,
	W =  90.000 deg,	P =   0.000 deg,	R =   90.000 deg
};
P[2421]{
   GP1:
	UF : 0, UT : 6,		CONFIG : 'N U T, 0, 0, 0',
	X =  411.188  mm,	Y =   -253.389  mm,	Z =   -229.016  mm,
	W =  90.000 deg,	P =   0.000 deg,	R =   90.000 deg
};
P[2422]{
   GP1:
	UF : 0, UT : 6,		CONFIG : 'N U T, 0, 0, 0',
	X =  409.734  mm,	Y =   -250.935  mm,	Z =   -229.104  mm,
	W =  90.000 deg,	P =   0.000 deg,	R =   90.000 deg
};
P[2423]{
   GP1:
	UF : 0, UT : 6,		CONFIG : 'N U T, 0, 0, 0',
	X =  409.177  mm,	Y =   -249.972  mm,	Z =   -229.105  mm,
	W =  90.000 deg,	P =   0.000 deg,	R =   90.000 deg
};
P[2424]{
   GP1:
	UF : 0, UT : 6,		CONFIG : 'N U T, 0, 0, 0',
	X =  408.714  mm,	Y =   -249.148  mm,	Z =   -229.076  mm,
	W =  90.000 deg,	P =   0.000 deg,	R =   90.000 deg
};
P[2425]{
   GP1:
	UF : 0, UT : 6,		CONFIG : 'N U T, 0, 0, 0',
	X =  407.999  mm,	Y =   -247.997  mm,	Z =   -229.199  mm,
	W =  90.000 deg,	P =   0.000 deg,	R =   90.000 deg
};
P[2426]{
   GP1:
	UF : 0, UT : 6,		CONFIG : 'N U T, 0, 0, 0',
	X =  406.765  mm,	Y =   -245.862  mm,	Z =   -229.203  mm,
	W =  90.000 deg,	P =   0.000 deg,	R =   90.000 deg
};
P[2427]{
   GP1:
	UF : 0, UT : 6,		CONFIG : 'N U T, 0, 0, 0',
	X =  405.991  mm,	Y =   -244.475  mm,	Z =   -229.136  mm,
	W =  90.000 deg,	P =   0.000 deg,	R =   90.000 deg
};
P[2428]{
   GP1:
	UF : 0, UT : 6,		CONFIG : 'N U T, 0, 0, 0',
	X =  405.666  mm,	Y =   -243.907  mm,	Z =   -229.130  mm,
	W =  90.000 deg,	P =   0.000 deg,	R =   90.000 deg
};
P[2429]{
   GP1:
	UF : 0, UT : 6,		CONFIG : 'N U T, 0, 0, 0',
	X =  404.932  mm,	Y =   -242.767  mm,	Z =   -229.314  mm,
	W =  90.000 deg,	P =   0.000 deg,	R =   90.000 deg
};
P[2430]{
   GP1:
	UF : 0, UT : 6,		CONFIG : 'N U T, 0, 0, 0',
	X =  403.024  mm,	Y =   -239.238  mm,	Z =   -228.999  mm,
	W =  90.000 deg,	P =   0.000 deg,	R =   90.000 deg
};
P[2431]{
   GP1:
	UF : 0, UT : 6,		CONFIG : 'N U T, 0, 0, 0',
	X =  402.586  mm,	Y =   -238.675  mm,	Z =   -229.272  mm,
	W =  90.000 deg,	P =   0.000 deg,	R =   90.000 deg
};
P[2432]{
   GP1:
	UF : 0, UT : 6,		CONFIG : 'N U T, 0, 0, 0',
	X =  401.645  mm,	Y =   -237.061  mm,	Z =   -229.294  mm,
	W =  90.000 deg,	P =   0.000 deg,	R =   90.000 deg
};
P[2433]{
   GP1:
	UF : 0, UT : 6,		CONFIG : 'N U T, 0, 0, 0',
	X =  401.321  mm,	Y =   -236.376  mm,	Z =   -229.122  mm,
	W =  90.000 deg,	P =   0.000 deg,	R =   90.000 deg
};
P[2434]{
   GP1:
	UF : 0, UT : 6,		CONFIG : 'N U T, 0, 0, 0',
	X =  399.953  mm,	Y =   -234.123  mm,	Z =   -229.283  mm,
	W =  90.000 deg,	P =   0.000 deg,	R =   90.000 deg
};
P[2435]{
   GP1:
	UF : 0, UT : 6,		CONFIG : 'N U T, 0, 0, 0',
	X =  398.972  mm,	Y =   -232.484  mm,	Z =   -229.369  mm,
	W =  90.000 deg,	P =   0.000 deg,	R =   90.000 deg
};
P[2436]{
   GP1:
	UF : 0, UT : 6,		CONFIG : 'N U T, 0, 0, 0',
	X =  398.386  mm,	Y =   -231.212  mm,	Z =   -229.008  mm,
	W =  90.000 deg,	P =   0.000 deg,	R =   90.000 deg
};
P[2437]{
   GP1:
	UF : 0, UT : 6,		CONFIG : 'N U T, 0, 0, 0',
	X =  397.998  mm,	Y =   -230.815  mm,	Z =   -229.394  mm,
	W =  90.000 deg,	P =   0.000 deg,	R =   90.000 deg
};
P[2438]{
   GP1:
	UF : 0, UT : 6,		CONFIG : 'N U T, 0, 0, 0',
	X =  397.806  mm,	Y =   -230.267  mm,	Z =   -229.092  mm,
	W =  90.000 deg,	P =   0.000 deg,	R =   90.000 deg
};
P[2439]{
   GP1:
	UF : 0, UT : 6,		CONFIG : 'N U T, 0, 0, 0',
	X =  396.917  mm,	Y =   -228.944  mm,	Z =   -229.397  mm,
	W =  90.000 deg,	P =   0.000 deg,	R =   90.000 deg
};
P[2440]{
   GP1:
	UF : 0, UT : 6,		CONFIG : 'N U T, 0, 0, 0',
	X =  395.878  mm,	Y =   -227.064  mm,	Z =   -229.283  mm,
	W =  90.000 deg,	P =   0.000 deg,	R =   90.000 deg
};
P[2441]{
   GP1:
	UF : 0, UT : 6,		CONFIG : 'N U T, 0, 0, 0',
	X =  394.159  mm,	Y =   -223.999  mm,	Z =   -229.159  mm,
	W =  90.000 deg,	P =   0.000 deg,	R =   90.000 deg
};
P[2442]{
   GP1:
	UF : 0, UT : 6,		CONFIG : 'N U T, 0, 0, 0',
	X =  393.246  mm,	Y =   -222.376  mm,	Z =   -229.100  mm,
	W =  90.000 deg,	P =   0.000 deg,	R =   90.000 deg
};
P[2443]{
   GP1:
	UF : 0, UT : 6,		CONFIG : 'N U T, 0, 0, 0',
	X =  392.703  mm,	Y =   -221.414  mm,	Z =   -229.068  mm,
	W =  90.000 deg,	P =   0.000 deg,	R =   90.000 deg
};
P[2444]{
   GP1:
	UF : 0, UT : 6,		CONFIG : 'N U T, 0, 0, 0',
	X =  392.343  mm,	Y =   -220.792  mm,	Z =   -229.072  mm,
	W =  90.000 deg,	P =   0.000 deg,	R =   90.000 deg
};
P[2445]{
   GP1:
	UF : 0, UT : 6,		CONFIG : 'N U T, 0, 0, 0',
	X =  391.884  mm,	Y =   -220.015  mm,	Z =   -229.099  mm,
	W =  90.000 deg,	P =   0.000 deg,	R =   90.000 deg
};
P[2446]{
   GP1:
	UF : 0, UT : 6,		CONFIG : 'N U T, 0, 0, 0',
	X =  391.414  mm,	Y =   -219.116  mm,	Z =   -228.977  mm,
	W =  90.000 deg,	P =   0.000 deg,	R =   90.000 deg
};
P[2447]{
   GP1:
	UF : 0, UT : 6,		CONFIG : 'N U T, 0, 0, 0',
	X =  391.023  mm,	Y =   -218.397  mm,	Z =   -228.920  mm,
	W =  90.000 deg,	P =   0.000 deg,	R =   90.000 deg
};
P[2448]{
   GP1:
	UF : 0, UT : 6,		CONFIG : 'N U T, 0, 0, 0',
	X =  390.432  mm,	Y =   -217.390  mm,	Z =   -228.944  mm,
	W =  90.000 deg,	P =   0.000 deg,	R =   90.000 deg
};
P[2449]{
   GP1:
	UF : 0, UT : 6,		CONFIG : 'N U T, 0, 0, 0',
	X =  389.910  mm,	Y =   -216.645  mm,	Z =   -229.164  mm,
	W =  90.000 deg,	P =   0.000 deg,	R =   90.000 deg
};
P[2450]{
   GP1:
	UF : 0, UT : 6,		CONFIG : 'N U T, 0, 0, 0',
	X =  389.526  mm,	Y =   -216.051  mm,	Z =   -229.265  mm,
	W =  90.000 deg,	P =   0.000 deg,	R =   90.000 deg
};
P[2451]{
   GP1:
	UF : 0, UT : 6,		CONFIG : 'N U T, 0, 0, 0',
	X =  388.512  mm,	Y =   -214.186  mm,	Z =   -229.114  mm,
	W =  90.000 deg,	P =   0.000 deg,	R =   90.000 deg
};
P[2452]{
   GP1:
	UF : 0, UT : 6,		CONFIG : 'N U T, 0, 0, 0',
	X =  387.628  mm,	Y =   -212.667  mm,	Z =   -229.130  mm,
	W =  90.000 deg,	P =   0.000 deg,	R =   90.000 deg
};
P[2453]{
   GP1:
	UF : 0, UT : 6,		CONFIG : 'N U T, 0, 0, 0',
	X =  386.693  mm,	Y =   -210.963  mm,	Z =   -229.011  mm,
	W =  90.000 deg,	P =   0.000 deg,	R =   90.000 deg
};
P[2454]{
   GP1:
	UF : 0, UT : 6,		CONFIG : 'N U T, 0, 0, 0',
	X =  386.103  mm,	Y =   -210.136  mm,	Z =   -229.285  mm,
	W =  90.000 deg,	P =   0.000 deg,	R =   90.000 deg
};
P[2455]{
   GP1:
	UF : 0, UT : 6,		CONFIG : 'N U T, 0, 0, 0',
	X =  383.499  mm,	Y =   -205.553  mm,	Z =   -229.181  mm,
	W =  90.000 deg,	P =   0.000 deg,	R =   90.000 deg
};
P[2456]{
   GP1:
	UF : 0, UT : 6,		CONFIG : 'N U T, 0, 0, 0',
	X =  382.900  mm,	Y =   -204.330  mm,	Z =   -228.921  mm,
	W =  90.000 deg,	P =   0.000 deg,	R =   90.000 deg
};
P[2457]{
   GP1:
	UF : 0, UT : 6,		CONFIG : 'N U T, 0, 0, 0',
	X =  381.676  mm,	Y =   -202.364  mm,	Z =   -229.136  mm,
	W =  90.000 deg,	P =   0.000 deg,	R =   90.000 deg
};
P[2458]{
   GP1:
	UF : 0, UT : 6,		CONFIG : 'N U T, 0, 0, 0',
	X =  380.976  mm,	Y =   -201.158  mm,	Z =   -229.147  mm,
	W =  90.000 deg,	P =   0.000 deg,	R =   90.000 deg
};
P[2459]{
   GP1:
	UF : 0, UT : 6,		CONFIG : 'N U T, 0, 0, 0',
	X =  380.274  mm,	Y =   -199.811  mm,	Z =   -228.963  mm,
	W =  90.000 deg,	P =   0.000 deg,	R =   90.000 deg
};
P[2460]{
   GP1:
	UF : 0, UT : 6,		CONFIG : 'N U T, 0, 0, 0',
	X =  377.720  mm,	Y =   -195.685  mm,	Z =   -229.380  mm,
	W =  90.000 deg,	P =   0.000 deg,	R =   90.000 deg
};
P[2461]{
   GP1:
	UF : 0, UT : 6,		CONFIG : 'N U T, 0, 0, 0',
	X =  375.953  mm,	Y =   -192.388  mm,	Z =   -229.048  mm,
	W =  90.000 deg,	P =   0.000 deg,	R =   90.000 deg
};
P[2462]{
   GP1:
	UF : 0, UT : 6,		CONFIG : 'N U T, 0, 0, 0',
	X =  375.420  mm,	Y =   -191.592  mm,	Z =   -229.227  mm,
	W =  90.000 deg,	P =   0.000 deg,	R =   90.000 deg
};
P[2463]{
   GP1:
	UF : 0, UT : 6,		CONFIG : 'N U T, 0, 0, 0',
	X =  374.933  mm,	Y =   -190.674  mm,	Z =   -229.121  mm,
	W =  90.000 deg,	P =   0.000 deg,	R =   90.000 deg
};
P[2464]{
   GP1:
	UF : 0, UT : 6,		CONFIG : 'N U T, 0, 0, 0',
	X =  374.400  mm,	Y =   -189.802  mm,	Z =   -229.194  mm,
	W =  90.000 deg,	P =   0.000 deg,	R =   90.000 deg
};
P[2465]{
   GP1:
	UF : 0, UT : 6,		CONFIG : 'N U T, 0, 0, 0',
	X =  369.502  mm,	Y =   -181.380  mm,	Z =   -229.277  mm,
	W =  90.000 deg,	P =   0.000 deg,	R =   90.000 deg
};
P[2466]{
   GP1:
	UF : 0, UT : 6,		CONFIG : 'N U T, 0, 0, 0',
	X =  369.014  mm,	Y =   -180.385  mm,	Z =   -229.071  mm,
	W =  90.000 deg,	P =   0.000 deg,	R =   90.000 deg
};
P[2467]{
   GP1:
	UF : 0, UT : 6,		CONFIG : 'N U T, 0, 0, 0',
	X =  368.552  mm,	Y =   -179.475  mm,	Z =   -228.914  mm,
	W =  90.000 deg,	P =   0.000 deg,	R =   90.000 deg
};
P[2468]{
   GP1:
	UF : 0, UT : 6,		CONFIG : 'N U T, 0, 0, 0',
	X =  367.344  mm,	Y =   -177.660  mm,	Z =   -229.305  mm,
	W =  90.000 deg,	P =   0.000 deg,	R =   90.000 deg
};
P[2469]{
   GP1:
	UF : 0, UT : 6,		CONFIG : 'N U T, 0, 0, 0',
	X =  366.654  mm,	Y =   -176.372  mm,	Z =   -229.172  mm,
	W =  90.000 deg,	P =   0.000 deg,	R =   90.000 deg
};
P[2470]{
   GP1:
	UF : 0, UT : 6,		CONFIG : 'N U T, 0, 0, 0',
	X =  366.221  mm,	Y =   -175.577  mm,	Z =   -229.109  mm,
	W =  90.000 deg,	P =   0.000 deg,	R =   90.000 deg
};
P[2471]{
   GP1:
	UF : 0, UT : 6,		CONFIG : 'N U T, 0, 0, 0',
	X =  364.962  mm,	Y =   -173.535  mm,	Z =   -229.303  mm,
	W =  90.000 deg,	P =   0.000 deg,	R =   90.000 deg
};
P[2472]{
   GP1:
	UF : 0, UT : 6,		CONFIG : 'N U T, 0, 0, 0',
	X =  363.745  mm,	Y =   -171.307  mm,	Z =   -229.132  mm,
	W =  90.000 deg,	P =   0.000 deg,	R =   90.000 deg
};
P[2473]{
   GP1:
	UF : 0, UT : 6,		CONFIG : 'N U T, 0, 0, 0',
	X =  361.424  mm,	Y =   -167.196  mm,	Z =   -229.008  mm,
	W =  90.000 deg,	P =   0.000 deg,	R =   90.000 deg
};
P[2474]{
   GP1:
	UF : 0, UT : 6,		CONFIG : 'N U T, 0, 0, 0',
	X =  360.902  mm,	Y =   -166.512  mm,	Z =   -229.316  mm,
	W =  90.000 deg,	P =   0.000 deg,	R =   90.000 deg
};
P[2475]{
   GP1:
	UF : 0, UT : 6,		CONFIG : 'N U T, 0, 0, 0',
	X =  359.293  mm,	Y =   -163.443  mm,	Z =   -228.921  mm,
	W =  90.000 deg,	P =   0.000 deg,	R =   90.000 deg
};
P[2476]{
   GP1:
	UF : 0, UT : 6,		CONFIG : 'N U T, 0, 0, 0',
	X =  358.671  mm,	Y =   -162.678  mm,	Z =   -229.358  mm,
	W =  90.000 deg,	P =   0.000 deg,	R =   90.000 deg
};
P[2477]{
   GP1:
	UF : 0, UT : 6,		CONFIG : 'N U T, 0, 0, 0',
	X =  358.193  mm,	Y =   -161.529  mm,	Z =   -228.908  mm,
	W =  90.000 deg,	P =   0.000 deg,	R =   90.000 deg
};
P[2478]{
   GP1:
	UF : 0, UT : 6,		CONFIG : 'N U T, 0, 0, 0',
	X =  357.698  mm,	Y =   -160.966  mm,	Z =   -229.319  mm,
	W =  90.000 deg,	P =   0.000 deg,	R =   90.000 deg
};
P[2479]{
   GP1:
	UF : 0, UT : 6,		CONFIG : 'N U T, 0, 0, 0',
	X =  357.250  mm,	Y =   -159.982  mm,	Z =   -229.029  mm,
	W =  90.000 deg,	P =   0.000 deg,	R =   90.000 deg
};
P[2480]{
   GP1:
	UF : 0, UT : 6,		CONFIG : 'N U T, 0, 0, 0',
	X =  356.806  mm,	Y =   -159.169  mm,	Z =   -228.968  mm,
	W =  90.000 deg,	P =   0.000 deg,	R =   90.000 deg
};
P[2481]{
   GP1:
	UF : 0, UT : 6,		CONFIG : 'N U T, 0, 0, 0',
	X =  355.410  mm,	Y =   -156.999  mm,	Z =   -229.314  mm,
	W =  90.000 deg,	P =   0.000 deg,	R =   90.000 deg
};
P[2482]{
   GP1:
	UF : 0, UT : 6,		CONFIG : 'N U T, 0, 0, 0',
	X =  355.082  mm,	Y =   -156.396  mm,	Z =   -229.263  mm,
	W =  90.000 deg,	P =   0.000 deg,	R =   90.000 deg
};
P[2483]{
   GP1:
	UF : 0, UT : 6,		CONFIG : 'N U T, 0, 0, 0',
	X =  354.891  mm,	Y =   -155.839  mm,	Z =   -228.947  mm,
	W =  90.000 deg,	P =   0.000 deg,	R =   90.000 deg
};
P[2484]{
   GP1:
	UF : 0, UT : 6,		CONFIG : 'N U T, 0, 0, 0',
	X =  354.242  mm,	Y =   -154.694  mm,	Z =   -228.920  mm,
	W =  90.000 deg,	P =   0.000 deg,	R =   90.000 deg
};
P[2485]{
   GP1:
	UF : 0, UT : 6,		CONFIG : 'N U T, 0, 0, 0',
	X =  351.819  mm,	Y =   -150.772  mm,	Z =   -229.303  mm,
	W =  90.000 deg,	P =   0.000 deg,	R =   90.000 deg
};
P[2486]{
   GP1:
	UF : 0, UT : 6,		CONFIG : 'N U T, 0, 0, 0',
	X =  351.460  mm,	Y =   -150.190  mm,	Z =   -229.360  mm,
	W =  90.000 deg,	P =   0.000 deg,	R =   90.000 deg
};
P[2487]{
   GP1:
	UF : 0, UT : 6,		CONFIG : 'N U T, 0, 0, 0',
	X =  350.986  mm,	Y =   -149.261  mm,	Z =   -229.209  mm,
	W =  90.000 deg,	P =   0.000 deg,	R =   90.000 deg
};
P[2488]{
   GP1:
	UF : 0, UT : 6,		CONFIG : 'N U T, 0, 0, 0',
	X =  350.745  mm,	Y =   -148.688  mm,	Z =   -228.991  mm,
	W =  90.000 deg,	P =   0.000 deg,	R =   90.000 deg
};
P[2489]{
   GP1:
	UF : 0, UT : 6,		CONFIG : 'N U T, 0, 0, 0',
	X =  349.738  mm,	Y =   -147.165  mm,	Z =   -229.297  mm,
	W =  90.000 deg,	P =   0.000 deg,	R =   90.000 deg
};
P[2490]{
   GP1:
	UF : 0, UT : 6,		CONFIG : 'N U T, 0, 0, 0',
	X =  348.949  mm,	Y =   -145.704  mm,	Z =   -229.167  mm,
	W =  90.000 deg,	P =   0.000 deg,	R =   90.000 deg
};
P[2491]{
   GP1:
	UF : 0, UT : 6,		CONFIG : 'N U T, 0, 0, 0',
	X =  347.927  mm,	Y =   -143.763  mm,	Z =   -228.925  mm,
	W =  90.000 deg,	P =   0.000 deg,	R =   90.000 deg
};
P[2492]{
   GP1:
	UF : 0, UT : 6,		CONFIG : 'N U T, 0, 0, 0',
	X =  345.924  mm,	Y =   -140.547  mm,	Z =   -229.283  mm,
	W =  90.000 deg,	P =   0.000 deg,	R =   90.000 deg
};
P[2493]{
   GP1:
	UF : 0, UT : 6,		CONFIG : 'N U T, 0, 0, 0',
	X =  345.302  mm,	Y =   -139.240  mm,	Z =   -228.960  mm,
	W =  90.000 deg,	P =   0.000 deg,	R =   90.000 deg
};
P[2494]{
   GP1:
	UF : 0, UT : 6,		CONFIG : 'N U T, 0, 0, 0',
	X =  344.718  mm,	Y =   -138.274  mm,	Z =   -229.024  mm,
	W =  90.000 deg,	P =   0.000 deg,	R =   90.000 deg
};
P[2495]{
   GP1:
	UF : 0, UT : 6,		CONFIG : 'N U T, 0, 0, 0',
	X =  344.309  mm,	Y =   -137.643  mm,	Z =   -229.080  mm,
	W =  90.000 deg,	P =   0.000 deg,	R =   90.000 deg
};
P[2496]{
   GP1:
	UF : 0, UT : 6,		CONFIG : 'N U T, 0, 0, 0',
	X =  343.786  mm,	Y =   -136.926  mm,	Z =   -229.111  mm,
	W =  90.000 deg,	P =   0.000 deg,	R =   90.000 deg
};
P[2497]{
   GP1:
	UF : 0, UT : 6,		CONFIG : 'N U T, 0, 0, 0',
	X =  341.416  mm,	Y =   -134.343  mm,	Z =   -229.257  mm,
	W =  90.000 deg,	P =   0.000 deg,	R =   90.000 deg
};
P[2498]{
   GP1:
	UF : 0, UT : 6,		CONFIG : 'N U T, 0, 0, 0',
	X =  340.794  mm,	Y =   -133.722  mm,	Z =   -229.090  mm,
	W =  90.000 deg,	P =   0.000 deg,	R =   90.000 deg
};
P[2499]{
   GP1:
	UF : 0, UT : 6,		CONFIG : 'N U T, 0, 0, 0',
	X =  338.813  mm,	Y =   -132.648  mm,	Z =   -229.325  mm,
	W =  90.000 deg,	P =   0.000 deg,	R =   90.000 deg
};
P[2500]{
   GP1:
	UF : 0, UT : 6,		CONFIG : 'N U T, 0, 0, 0',
	X =  336.730  mm,	Y =   -131.730  mm,	Z =   -229.095  mm,
	W =  90.000 deg,	P =   0.000 deg,	R =   90.000 deg
};
P[2501]{
   GP1:
	UF : 0, UT : 6,		CONFIG : 'N U T, 0, 0, 0',
	X =  335.243  mm,	Y =   -131.534  mm,	Z =   -229.291  mm,
	W =  90.000 deg,	P =   0.000 deg,	R =   90.000 deg
};
P[2502]{
   GP1:
	UF : 0, UT : 6,		CONFIG : 'N U T, 0, 0, 0',
	X =  334.335  mm,	Y =   -131.427  mm,	Z =   -229.352  mm,
	W =  90.000 deg,	P =   0.000 deg,	R =   90.000 deg
};
P[2503]{
   GP1:
	UF : 0, UT : 6,		CONFIG : 'N U T, 0, 0, 0',
	X =  332.692  mm,	Y =   -131.384  mm,	Z =   -229.229  mm,
	W =  90.000 deg,	P =   0.000 deg,	R =   90.000 deg
};
P[2504]{
   GP1:
	UF : 0, UT : 6,		CONFIG : 'N U T, 0, 0, 0',
	X =  331.744  mm,	Y =   -131.350  mm,	Z =   -229.052  mm,
	W =  90.000 deg,	P =   0.000 deg,	R =   90.000 deg
};
P[2505]{
   GP1:
	UF : 0, UT : 6,		CONFIG : 'N U T, 0, 0, 0',
	X =  327.919  mm,	Y =   -132.483  mm,	Z =   -228.957  mm,
	W =  90.000 deg,	P =   0.000 deg,	R =   90.000 deg
};
P[2506]{
   GP1:
	UF : 0, UT : 6,		CONFIG : 'N U T, 0, 0, 0',
	X =  325.434  mm,	Y =   -133.800  mm,	Z =   -229.001  mm,
	W =  90.000 deg,	P =   0.000 deg,	R =   90.000 deg
};
P[2507]{
   GP1:
	UF : 0, UT : 6,		CONFIG : 'N U T, 0, 0, 0',
	X =  324.678  mm,	Y =   -134.226  mm,	Z =   -228.975  mm,
	W =  90.000 deg,	P =   0.000 deg,	R =   90.000 deg
};
P[2508]{
   GP1:
	UF : 0, UT : 6,		CONFIG : 'N U T, 0, 0, 0',
	X =  323.692  mm,	Y =   -134.879  mm,	Z =   -229.176  mm,
	W =  90.000 deg,	P =   0.000 deg,	R =   90.000 deg
};
P[2509]{
   GP1:
	UF : 0, UT : 6,		CONFIG : 'N U T, 0, 0, 0',
	X =  320.956  mm,	Y =   -136.352  mm,	Z =   -228.917  mm,
	W =  90.000 deg,	P =   0.000 deg,	R =   90.000 deg
};
P[2510]{
   GP1:
	UF : 0, UT : 6,		CONFIG : 'N U T, 0, 0, 0',
	X =  319.628  mm,	Y =   -137.249  mm,	Z =   -229.235  mm,
	W =  90.000 deg,	P =   0.000 deg,	R =   90.000 deg
};
P[2511]{
   GP1:
	UF : 0, UT : 6,		CONFIG : 'N U T, 0, 0, 0',
	X =  317.845  mm,	Y =   -138.271  mm,	Z =   -229.215  mm,
	W =  90.000 deg,	P =   0.000 deg,	R =   90.000 deg
};
P[2512]{
   GP1:
	UF : 0, UT : 6,		CONFIG : 'N U T, 0, 0, 0',
	X =  316.218  mm,	Y =   -139.111  mm,	Z =   -228.975  mm,
	W =  90.000 deg,	P =   0.000 deg,	R =   90.000 deg
};
P[2513]{
   GP1:
	UF : 0, UT : 6,		CONFIG : 'N U T, 0, 0, 0',
	X =  315.305  mm,	Y =   -139.769  mm,	Z =   -229.294  mm,
	W =  90.000 deg,	P =   0.000 deg,	R =   90.000 deg
};
P[2514]{
   GP1:
	UF : 0, UT : 6,		CONFIG : 'N U T, 0, 0, 0',
	X =  314.621  mm,	Y =   -140.104  mm,	Z =   -229.146  mm,
	W =  90.000 deg,	P =   0.000 deg,	R =   90.000 deg
};
P[2515]{
   GP1:
	UF : 0, UT : 6,		CONFIG : 'N U T, 0, 0, 0',
	X =  314.061  mm,	Y =   -140.440  mm,	Z =   -229.178  mm,
	W =  90.000 deg,	P =   0.000 deg,	R =   90.000 deg
};
P[2516]{
   GP1:
	UF : 0, UT : 6,		CONFIG : 'N U T, 0, 0, 0',
	X =  313.031  mm,	Y =   -141.121  mm,	Z =   -229.389  mm,
	W =  90.000 deg,	P =   0.000 deg,	R =   90.000 deg
};
P[2517]{
   GP1:
	UF : 0, UT : 6,		CONFIG : 'N U T, 0, 0, 0',
	X =  310.536  mm,	Y =   -142.458  mm,	Z =   -229.136  mm,
	W =  90.000 deg,	P =   0.000 deg,	R =   90.000 deg
};
P[2518]{
   GP1:
	UF : 0, UT : 6,		CONFIG : 'N U T, 0, 0, 0',
	X =  309.932  mm,	Y =   -142.770  mm,	Z =   -229.045  mm,
	W =  90.000 deg,	P =   0.000 deg,	R =   90.000 deg
};
P[2519]{
   GP1:
	UF : 0, UT : 6,		CONFIG : 'N U T, 0, 0, 0',
	X =  308.389  mm,	Y =   -143.609  mm,	Z =   -228.922  mm,
	W =  90.000 deg,	P =   0.000 deg,	R =   90.000 deg
};
P[2520]{
   GP1:
	UF : 0, UT : 6,		CONFIG : 'N U T, 0, 0, 0',
	X =  306.991  mm,	Y =   -144.512  mm,	Z =   -229.151  mm,
	W =  90.000 deg,	P =   0.000 deg,	R =   90.000 deg
};
P[2521]{
   GP1:
	UF : 0, UT : 6,		CONFIG : 'N U T, 0, 0, 0',
	X =  305.259  mm,	Y =   -145.593  mm,	Z =   -229.350  mm,
	W =  90.000 deg,	P =   0.000 deg,	R =   90.000 deg
};
P[2522]{
   GP1:
	UF : 0, UT : 6,		CONFIG : 'N U T, 0, 0, 0',
	X =  302.827  mm,	Y =   -146.983  mm,	Z =   -229.317  mm,
	W =  90.000 deg,	P =   0.000 deg,	R =   90.000 deg
};
P[2523]{
   GP1:
	UF : 0, UT : 6,		CONFIG : 'N U T, 0, 0, 0',
	X =  297.144  mm,	Y =   -150.180  mm,	Z =   -229.111  mm,
	W =  90.000 deg,	P =   0.000 deg,	R =   90.000 deg
};
P[2524]{
   GP1:
	UF : 0, UT : 6,		CONFIG : 'N U T, 0, 0, 0',
	X =  296.108  mm,	Y =   -150.727  mm,	Z =   -228.986  mm,
	W =  90.000 deg,	P =   0.000 deg,	R =   90.000 deg
};
P[2525]{
   GP1:
	UF : 0, UT : 6,		CONFIG : 'N U T, 0, 0, 0',
	X =  295.398  mm,	Y =   -151.259  mm,	Z =   -229.283  mm,
	W =  90.000 deg,	P =   0.000 deg,	R =   90.000 deg
};
P[2526]{
   GP1:
	UF : 0, UT : 6,		CONFIG : 'N U T, 0, 0, 0',
	X =  291.372  mm,	Y =   -153.473  mm,	Z =   -229.012  mm,
	W =  90.000 deg,	P =   0.000 deg,	R =   90.000 deg
};
P[2527]{
   GP1:
	UF : 0, UT : 6,		CONFIG : 'N U T, 0, 0, 0',
	X =  290.468  mm,	Y =   -153.951  mm,	Z =   -228.907  mm,
	W =  90.000 deg,	P =   0.000 deg,	R =   90.000 deg
};
P[2528]{
   GP1:
	UF : 0, UT : 6,		CONFIG : 'N U T, 0, 0, 0',
	X =  288.482  mm,	Y =   -155.117  mm,	Z =   -228.954  mm,
	W =  90.000 deg,	P =   0.000 deg,	R =   90.000 deg
};
P[2529]{
   GP1:
	UF : 0, UT : 6,		CONFIG : 'N U T, 0, 0, 0',
	X =  287.721  mm,	Y =   -155.703  mm,	Z =   -229.309  mm,
	W =  90.000 deg,	P =   0.000 deg,	R =   90.000 deg
};
P[2530]{
   GP1:
	UF : 0, UT : 6,		CONFIG : 'N U T, 0, 0, 0',
	X =  287.207  mm,	Y =   -155.830  mm,	Z =   -228.898  mm,
	W =  90.000 deg,	P =   0.000 deg,	R =   90.000 deg
};
P[2531]{
   GP1:
	UF : 0, UT : 6,		CONFIG : 'N U T, 0, 0, 0',
	X =  283.909  mm,	Y =   -157.872  mm,	Z =   -229.230  mm,
	W =  90.000 deg,	P =   0.000 deg,	R =   90.000 deg
};
P[2532]{
   GP1:
	UF : 0, UT : 6,		CONFIG : 'N U T, 0, 0, 0',
	X =  282.884  mm,	Y =   -158.410  mm,	Z =   -229.103  mm,
	W =  90.000 deg,	P =   0.000 deg,	R =   90.000 deg
};
P[2533]{
   GP1:
	UF : 0, UT : 6,		CONFIG : 'N U T, 0, 0, 0',
	X =  281.669  mm,	Y =   -159.176  mm,	Z =   -229.259  mm,
	W =  90.000 deg,	P =   0.000 deg,	R =   90.000 deg
};
P[2534]{
   GP1:
	UF : 0, UT : 6,		CONFIG : 'N U T, 0, 0, 0',
	X =  280.516  mm,	Y =   -159.746  mm,	Z =   -229.025  mm,
	W =  90.000 deg,	P =   0.000 deg,	R =   90.000 deg
};
P[2535]{
   GP1:
	UF : 0, UT : 6,		CONFIG : 'N U T, 0, 0, 0',
	X =  279.591  mm,	Y =   -160.374  mm,	Z =   -229.254  mm,
	W =  90.000 deg,	P =   0.000 deg,	R =   90.000 deg
};
P[2536]{
   GP1:
	UF : 0, UT : 6,		CONFIG : 'N U T, 0, 0, 0',
	X =  278.873  mm,	Y =   -160.783  mm,	Z =   -229.239  mm,
	W =  90.000 deg,	P =   0.000 deg,	R =   90.000 deg
};
P[2537]{
   GP1:
	UF : 0, UT : 6,		CONFIG : 'N U T, 0, 0, 0',
	X =  277.132  mm,	Y =   -161.661  mm,	Z =   -228.931  mm,
	W =  90.000 deg,	P =   0.000 deg,	R =   90.000 deg
};
P[2538]{
   GP1:
	UF : 0, UT : 6,		CONFIG : 'N U T, 0, 0, 0',
	X =  272.581  mm,	Y =   -164.357  mm,	Z =   -229.099  mm,
	W =  90.000 deg,	P =   0.000 deg,	R =   90.000 deg
};
P[2539]{
   GP1:
	UF : 0, UT : 6,		CONFIG : 'N U T, 0, 0, 0',
	X =  271.962  mm,	Y =   -164.648  mm,	Z =   -228.937  mm,
	W =  90.000 deg,	P =   0.000 deg,	R =   90.000 deg
};
P[2540]{
   GP1:
	UF : 0, UT : 6,		CONFIG : 'N U T, 0, 0, 0',
	X =  269.685  mm,	Y =   -166.005  mm,	Z =   -229.040  mm,
	W =  90.000 deg,	P =   0.000 deg,	R =   90.000 deg
};
P[2541]{
   GP1:
	UF : 0, UT : 6,		CONFIG : 'N U T, 0, 0, 0',
	X =  268.803  mm,	Y =   -166.464  mm,	Z =   -228.916  mm,
	W =  90.000 deg,	P =   0.000 deg,	R =   90.000 deg
};
P[2542]{
   GP1:
	UF : 0, UT : 6,		CONFIG : 'N U T, 0, 0, 0',
	X =  267.101  mm,	Y =   -167.640  mm,	Z =   -229.386  mm,
	W =  90.000 deg,	P =   0.000 deg,	R =   90.000 deg
};
P[2543]{
   GP1:
	UF : 0, UT : 6,		CONFIG : 'N U T, 0, 0, 0',
	X =  265.673  mm,	Y =   -168.341  mm,	Z =   -229.084  mm,
	W =  90.000 deg,	P =   0.000 deg,	R =   90.000 deg
};
P[2544]{
   GP1:
	UF : 0, UT : 6,		CONFIG : 'N U T, 0, 0, 0',
	X =  264.446  mm,	Y =   -169.175  mm,	Z =   -229.390  mm,
	W =  90.000 deg,	P =   0.000 deg,	R =   90.000 deg
};
P[2545]{
   GP1:
	UF : 0, UT : 6,		CONFIG : 'N U T, 0, 0, 0',
	X =  262.695  mm,	Y =   -170.111  mm,	Z =   -229.207  mm,
	W =  90.000 deg,	P =   0.000 deg,	R =   90.000 deg
};
P[2546]{
   GP1:
	UF : 0, UT : 6,		CONFIG : 'N U T, 0, 0, 0',
	X =  260.304  mm,	Y =   -171.417  mm,	Z =   -229.029  mm,
	W =  90.000 deg,	P =   0.000 deg,	R =   90.000 deg
};
P[2547]{
   GP1:
	UF : 0, UT : 6,		CONFIG : 'N U T, 0, 0, 0',
	X =  259.025  mm,	Y =   -172.228  mm,	Z =   -229.202  mm,
	W =  90.000 deg,	P =   0.000 deg,	R =   90.000 deg
};
P[2548]{
   GP1:
	UF : 0, UT : 6,		CONFIG : 'N U T, 0, 0, 0',
	X =  258.315  mm,	Y =   -172.611  mm,	Z =   -229.137  mm,
	W =  90.000 deg,	P =   0.000 deg,	R =   90.000 deg
};
P[2549]{
   GP1:
	UF : 0, UT : 6,		CONFIG : 'N U T, 0, 0, 0',
	X =  257.125  mm,	Y =   -173.228  mm,	Z =   -228.968  mm,
	W =  90.000 deg,	P =   0.000 deg,	R =   90.000 deg
};
P[2550]{
   GP1:
	UF : 0, UT : 6,		CONFIG : 'N U T, 0, 0, 0',
	X =  255.879  mm,	Y =   -174.012  mm,	Z =   -229.127  mm,
	W =  90.000 deg,	P =   0.000 deg,	R =   90.000 deg
};
P[2551]{
   GP1:
	UF : 0, UT : 6,		CONFIG : 'N U T, 0, 0, 0',
	X =  255.037  mm,	Y =   -174.562  mm,	Z =   -229.280  mm,
	W =  90.000 deg,	P =   0.000 deg,	R =   90.000 deg
};
P[2552]{
   GP1:
	UF : 0, UT : 6,		CONFIG : 'N U T, 0, 0, 0',
	X =  254.296  mm,	Y =   -174.964  mm,	Z =   -229.215  mm,
	W =  90.000 deg,	P =   0.000 deg,	R =   90.000 deg
};
P[2553]{
   GP1:
	UF : 0, UT : 6,		CONFIG : 'N U T, 0, 0, 0',
	X =  247.141  mm,	Y =   -179.142  mm,	Z =   -229.329  mm,
	W =  90.000 deg,	P =   0.000 deg,	R =   90.000 deg
};
P[2554]{
   GP1:
	UF : 0, UT : 6,		CONFIG : 'N U T, 0, 0, 0',
	X =  246.425  mm,	Y =   -179.493  mm,	Z =   -229.177  mm,
	W =  90.000 deg,	P =   0.000 deg,	R =   90.000 deg
};
P[2555]{
   GP1:
	UF : 0, UT : 6,		CONFIG : 'N U T, 0, 0, 0',
	X =  244.691  mm,	Y =   -180.577  mm,	Z =   -229.381  mm,
	W =  90.000 deg,	P =   0.000 deg,	R =   90.000 deg
};
P[2556]{
   GP1:
	UF : 0, UT : 6,		CONFIG : 'N U T, 0, 0, 0',
	X =  241.032  mm,	Y =   -182.637  mm,	Z =   -229.253  mm,
	W =  90.000 deg,	P =   0.000 deg,	R =   90.000 deg
};
P[2557]{
   GP1:
	UF : 0, UT : 6,		CONFIG : 'N U T, 0, 0, 0',
	X =  238.558  mm,	Y =   -184.045  mm,	Z =   -229.203  mm,
	W =  90.000 deg,	P =   0.000 deg,	R =   90.000 deg
};
P[2558]{
   GP1:
	UF : 0, UT : 6,		CONFIG : 'N U T, 0, 0, 0',
	X =  236.214  mm,	Y =   -185.276  mm,	Z =   -228.904  mm,
	W =  90.000 deg,	P =   0.000 deg,	R =   90.000 deg
};
P[2559]{
   GP1:
	UF : 0, UT : 6,		CONFIG : 'N U T, 0, 0, 0',
	X =  235.499  mm,	Y =   -185.688  mm,	Z =   -228.904  mm,
	W =  90.000 deg,	P =   0.000 deg,	R =   90.000 deg
};
P[2560]{
   GP1:
	UF : 0, UT : 6,		CONFIG : 'N U T, 0, 0, 0',
	X =  234.946  mm,	Y =   -186.086  mm,	Z =   -229.091  mm,
	W =  90.000 deg,	P =   0.000 deg,	R =   90.000 deg
};
P[2561]{
   GP1:
	UF : 0, UT : 6,		CONFIG : 'N U T, 0, 0, 0',
	X =  233.239  mm,	Y =   -187.134  mm,	Z =   -229.243  mm,
	W =  90.000 deg,	P =   0.000 deg,	R =   90.000 deg
};
P[2562]{
   GP1:
	UF : 0, UT : 6,		CONFIG : 'N U T, 0, 0, 0',
	X =  232.142  mm,	Y =   -187.741  mm,	Z =   -229.180  mm,
	W =  90.000 deg,	P =   0.000 deg,	R =   90.000 deg
};
P[2563]{
   GP1:
	UF : 0, UT : 6,		CONFIG : 'N U T, 0, 0, 0',
	X =  230.352  mm,	Y =   -188.703  mm,	Z =   -229.009  mm,
	W =  90.000 deg,	P =   0.000 deg,	R =   90.000 deg
};
P[2564]{
   GP1:
	UF : 0, UT : 6,		CONFIG : 'N U T, 0, 0, 0',
	X =  229.763  mm,	Y =   -189.187  mm,	Z =   -229.358  mm,
	W =  90.000 deg,	P =   0.000 deg,	R =   90.000 deg
};
P[2565]{
   GP1:
	UF : 0, UT : 6,		CONFIG : 'N U T, 0, 0, 0',
	X =  227.727  mm,	Y =   -190.279  mm,	Z =   -229.154  mm,
	W =  90.000 deg,	P =   0.000 deg,	R =   90.000 deg
};
P[2566]{
   GP1:
	UF : 0, UT : 6,		CONFIG : 'N U T, 0, 0, 0',
	X =  226.556  mm,	Y =   -190.885  mm,	Z =   -228.984  mm,
	W =  90.000 deg,	P =   0.000 deg,	R =   90.000 deg
};
P[2567]{
   GP1:
	UF : 0, UT : 6,		CONFIG : 'N U T, 0, 0, 0',
	X =  225.032  mm,	Y =   -191.934  mm,	Z =   -229.392  mm,
	W =  90.000 deg,	P =   0.000 deg,	R =   90.000 deg
};
P[2568]{
   GP1:
	UF : 0, UT : 6,		CONFIG : 'N U T, 0, 0, 0',
	X =  222.872  mm,	Y =   -193.076  mm,	Z =   -229.138  mm,
	W =  90.000 deg,	P =   0.000 deg,	R =   90.000 deg
};
P[2569]{
   GP1:
	UF : 0, UT : 6,		CONFIG : 'N U T, 0, 0, 0',
	X =  221.102  mm,	Y =   -194.047  mm,	Z =   -229.016  mm,
	W =  90.000 deg,	P =   0.000 deg,	R =   90.000 deg
};
P[2570]{
   GP1:
	UF : 0, UT : 6,		CONFIG : 'N U T, 0, 0, 0',
	X =  216.285  mm,	Y =   -196.911  mm,	Z =   -229.216  mm,
	W =  90.000 deg,	P =   0.000 deg,	R =   90.000 deg
};
P[2571]{
   GP1:
	UF : 0, UT : 6,		CONFIG : 'N U T, 0, 0, 0',
	X =  214.744  mm,	Y =   -197.854  mm,	Z =   -229.344  mm,
	W =  90.000 deg,	P =   0.000 deg,	R =   90.000 deg
};
P[2572]{
   GP1:
	UF : 0, UT : 6,		CONFIG : 'N U T, 0, 0, 0',
	X =  214.214  mm,	Y =   -198.003  mm,	Z =   -228.965  mm,
	W =  90.000 deg,	P =   0.000 deg,	R =   90.000 deg
};
P[2573]{
   GP1:
	UF : 0, UT : 6,		CONFIG : 'N U T, 0, 0, 0',
	X =  212.345  mm,	Y =   -199.164  mm,	Z =   -229.162  mm,
	W =  90.000 deg,	P =   0.000 deg,	R =   90.000 deg
};
P[2574]{
   GP1:
	UF : 0, UT : 6,		CONFIG : 'N U T, 0, 0, 0',
	X =  209.743  mm,	Y =   -200.581  mm,	Z =   -228.957  mm,
	W =  90.000 deg,	P =   0.000 deg,	R =   90.000 deg
};
P[2575]{
   GP1:
	UF : 0, UT : 6,		CONFIG : 'N U T, 0, 0, 0',
	X =  207.414  mm,	Y =   -201.979  mm,	Z =   -229.086  mm,
	W =  90.000 deg,	P =   0.000 deg,	R =   90.000 deg
};
P[2576]{
   GP1:
	UF : 0, UT : 6,		CONFIG : 'N U T, 0, 0, 0',
	X =  206.481  mm,	Y =   -202.501  mm,	Z =   -229.044  mm,
	W =  90.000 deg,	P =   0.000 deg,	R =   90.000 deg
};
P[2577]{
   GP1:
	UF : 0, UT : 6,		CONFIG : 'N U T, 0, 0, 0',
	X =  205.696  mm,	Y =   -203.066  mm,	Z =   -229.317  mm,
	W =  90.000 deg,	P =   0.000 deg,	R =   90.000 deg
};
P[2578]{
   GP1:
	UF : 0, UT : 6,		CONFIG : 'N U T, 0, 0, 0',
	X =  203.349  mm,	Y =   -204.257  mm,	Z =   -228.915  mm,
	W =  90.000 deg,	P =   0.000 deg,	R =   90.000 deg
};
P[2579]{
   GP1:
	UF : 0, UT : 6,		CONFIG : 'N U T, 0, 0, 0',
	X =  202.165  mm,	Y =   -205.106  mm,	Z =   -229.318  mm,
	W =  90.000 deg,	P =   0.000 deg,	R =   90.000 deg
};
P[2580]{
   GP1:
	UF : 0, UT : 6,		CONFIG : 'N U T, 0, 0, 0',
	X =  199.571  mm,	Y =   -206.515  mm,	Z =   -229.102  mm,
	W =  90.000 deg,	P =   0.000 deg,	R =   90.000 deg
};
P[2581]{
   GP1:
	UF : 0, UT : 6,		CONFIG : 'N U T, 0, 0, 0',
	X =  198.648  mm,	Y =   -206.965  mm,	Z =   -228.903  mm,
	W =  90.000 deg,	P =   0.000 deg,	R =   90.000 deg
};
P[2582]{
   GP1:
	UF : 0, UT : 6,		CONFIG : 'N U T, 0, 0, 0',
	X =  197.256  mm,	Y =   -207.858  mm,	Z =   -229.119  mm,
	W =  90.000 deg,	P =   0.000 deg,	R =   90.000 deg
};
P[2583]{
   GP1:
	UF : 0, UT : 6,		CONFIG : 'N U T, 0, 0, 0',
	X =  195.995  mm,	Y =   -208.663  mm,	Z =   -229.305  mm,
	W =  90.000 deg,	P =   0.000 deg,	R =   90.000 deg
};
P[2584]{
   GP1:
	UF : 0, UT : 6,		CONFIG : 'N U T, 0, 0, 0',
	X =  194.142  mm,	Y =   -209.730  mm,	Z =   -229.298  mm,
	W =  90.000 deg,	P =   0.000 deg,	R =   90.000 deg
};
P[2585]{
   GP1:
	UF : 0, UT : 6,		CONFIG : 'N U T, 0, 0, 0',
	X =  193.498  mm,	Y =   -210.076  mm,	Z =   -229.236  mm,
	W =  90.000 deg,	P =   0.000 deg,	R =   90.000 deg
};
P[2586]{
   GP1:
	UF : 0, UT : 6,		CONFIG : 'N U T, 0, 0, 0',
	X =  192.707  mm,	Y =   -210.422  mm,	Z =   -228.968  mm,
	W =  90.000 deg,	P =   0.000 deg,	R =   90.000 deg
};
P[2587]{
   GP1:
	UF : 0, UT : 6,		CONFIG : 'N U T, 0, 0, 0',
	X =  191.655  mm,	Y =   -211.190  mm,	Z =   -229.357  mm,
	W =  90.000 deg,	P =   0.000 deg,	R =   90.000 deg
};
P[2588]{
   GP1:
	UF : 0, UT : 6,		CONFIG : 'N U T, 0, 0, 0',
	X =  190.265  mm,	Y =   -211.907  mm,	Z =   -229.149  mm,
	W =  90.000 deg,	P =   0.000 deg,	R =   90.000 deg
};
P[2589]{
   GP1:
	UF : 0, UT : 6,		CONFIG : 'N U T, 0, 0, 0',
	X =  188.774  mm,	Y =   -212.833  mm,	Z =   -229.306  mm,
	W =  90.000 deg,	P =   0.000 deg,	R =   90.000 deg
};
P[2590]{
   GP1:
	UF : 0, UT : 6,		CONFIG : 'N U T, 0, 0, 0',
	X =  188.226  mm,	Y =   -212.997  mm,	Z =   -228.937  mm,
	W =  90.000 deg,	P =   0.000 deg,	R =   90.000 deg
};
P[2591]{
   GP1:
	UF : 0, UT : 6,		CONFIG : 'N U T, 0, 0, 0',
	X =  187.712  mm,	Y =   -213.472  mm,	Z =   -229.370  mm,
	W =  90.000 deg,	P =   0.000 deg,	R =   90.000 deg
};
P[2592]{
   GP1:
	UF : 0, UT : 6,		CONFIG : 'N U T, 0, 0, 0',
	X =  187.113  mm,	Y =   -213.632  mm,	Z =   -228.918  mm,
	W =  90.000 deg,	P =   0.000 deg,	R =   90.000 deg
};
P[2593]{
   GP1:
	UF : 0, UT : 6,		CONFIG : 'N U T, 0, 0, 0',
	X =  179.247  mm,	Y =   -218.211  mm,	Z =   -229.007  mm,
	W =  90.000 deg,	P =   0.000 deg,	R =   90.000 deg
};
P[2594]{
   GP1:
	UF : 0, UT : 6,		CONFIG : 'N U T, 0, 0, 0',
	X =  178.236  mm,	Y =   -218.853  mm,	Z =   -229.151  mm,
	W =  90.000 deg,	P =   0.000 deg,	R =   90.000 deg
};
P[2595]{
   GP1:
	UF : 0, UT : 6,		CONFIG : 'N U T, 0, 0, 0',
	X =  176.149  mm,	Y =   -219.999  mm,	Z =   -229.009  mm,
	W =  90.000 deg,	P =   0.000 deg,	R =   90.000 deg
};
P[2596]{
   GP1:
	UF : 0, UT : 6,		CONFIG : 'N U T, 0, 0, 0',
	X =  175.171  mm,	Y =   -220.659  mm,	Z =   -229.239  mm,
	W =  90.000 deg,	P =   0.000 deg,	R =   90.000 deg
};
P[2597]{
   GP1:
	UF : 0, UT : 6,		CONFIG : 'N U T, 0, 0, 0',
	X =  174.405  mm,	Y =   -221.102  mm,	Z =   -229.240  mm,
	W =  90.000 deg,	P =   0.000 deg,	R =   90.000 deg
};
P[2598]{
   GP1:
	UF : 0, UT : 6,		CONFIG : 'N U T, 0, 0, 0',
	X =  173.550  mm,	Y =   -221.620  mm,	Z =   -229.298  mm,
	W =  90.000 deg,	P =   0.000 deg,	R =   90.000 deg
};
P[2599]{
   GP1:
	UF : 0, UT : 6,		CONFIG : 'N U T, 0, 0, 0',
	X =  172.564  mm,	Y =   -222.049  mm,	Z =   -228.959  mm,
	W =  90.000 deg,	P =   0.000 deg,	R =   90.000 deg
};
P[2600]{
   GP1:
	UF : 0, UT : 6,		CONFIG : 'N U T, 0, 0, 0',
	X =  171.690  mm,	Y =   -222.623  mm,	Z =   -229.126  mm,
	W =  90.000 deg,	P =   0.000 deg,	R =   90.000 deg
};
P[2601]{
   GP1:
	UF : 0, UT : 6,		CONFIG : 'N U T, 0, 0, 0',
	X =  170.098  mm,	Y =   -223.466  mm,	Z =   -228.943  mm,
	W =  90.000 deg,	P =   0.000 deg,	R =   90.000 deg
};
P[2602]{
   GP1:
	UF : 0, UT : 6,		CONFIG : 'N U T, 0, 0, 0',
	X =  169.242  mm,	Y =   -224.096  mm,	Z =   -229.271  mm,
	W =  90.000 deg,	P =   0.000 deg,	R =   90.000 deg
};
P[2603]{
   GP1:
	UF : 0, UT : 6,		CONFIG : 'N U T, 0, 0, 0',
	X =  168.207  mm,	Y =   -224.625  mm,	Z =   -229.105  mm,
	W =  90.000 deg,	P =   0.000 deg,	R =   90.000 deg
};
P[2604]{
   GP1:
	UF : 0, UT : 6,		CONFIG : 'N U T, 0, 0, 0',
	X =  166.042  mm,	Y =   -225.988  mm,	Z =   -229.380  mm,
	W =  90.000 deg,	P =   0.000 deg,	R =   90.000 deg
};
P[2605]{
   GP1:
	UF : 0, UT : 6,		CONFIG : 'N U T, 0, 0, 0',
	X =  165.234  mm,	Y =   -226.460  mm,	Z =   -229.392  mm,
	W =  90.000 deg,	P =   0.000 deg,	R =   90.000 deg
};
P[2606]{
   GP1:
	UF : 0, UT : 6,		CONFIG : 'N U T, 0, 0, 0',
	X =  164.582  mm,	Y =   -226.784  mm,	Z =   -229.266  mm,
	W =  90.000 deg,	P =   0.000 deg,	R =   90.000 deg
};
P[2607]{
   GP1:
	UF : 0, UT : 6,		CONFIG : 'N U T, 0, 0, 0',
	X =  163.996  mm,	Y =   -227.056  mm,	Z =   -229.104  mm,
	W =  90.000 deg,	P =   0.000 deg,	R =   90.000 deg
};
P[2608]{
   GP1:
	UF : 0, UT : 6,		CONFIG : 'N U T, 0, 0, 0',
	X =  163.368  mm,	Y =   -227.467  mm,	Z =   -229.220  mm,
	W =  90.000 deg,	P =   0.000 deg,	R =   90.000 deg
};
P[2609]{
   GP1:
	UF : 0, UT : 6,		CONFIG : 'N U T, 0, 0, 0',
	X =  162.552  mm,	Y =   -227.887  mm,	Z =   -229.099  mm,
	W =  90.000 deg,	P =   0.000 deg,	R =   90.000 deg
};
P[2610]{
   GP1:
	UF : 0, UT : 6,		CONFIG : 'N U T, 0, 0, 0',
	X =  160.891  mm,	Y =   -228.936  mm,	Z =   -229.316  mm,
	W =  90.000 deg,	P =   0.000 deg,	R =   90.000 deg
};
P[2611]{
   GP1:
	UF : 0, UT : 6,		CONFIG : 'N U T, 0, 0, 0',
	X =  160.194  mm,	Y =   -229.203  mm,	Z =   -228.988  mm,
	W =  90.000 deg,	P =   0.000 deg,	R =   90.000 deg
};
P[2612]{
   GP1:
	UF : 0, UT : 6,		CONFIG : 'N U T, 0, 0, 0',
	X =  159.541  mm,	Y =   -229.604  mm,	Z =   -229.046  mm,
	W =  90.000 deg,	P =   0.000 deg,	R =   90.000 deg
};
P[2613]{
   GP1:
	UF : 0, UT : 6,		CONFIG : 'N U T, 0, 0, 0',
	X =  158.388  mm,	Y =   -230.238  mm,	Z =   -228.966  mm,
	W =  90.000 deg,	P =   0.000 deg,	R =   90.000 deg
};
P[2614]{
   GP1:
	UF : 0, UT : 6,		CONFIG : 'N U T, 0, 0, 0',
	X =  157.785  mm,	Y =   -230.606  mm,	Z =   -229.016  mm,
	W =  90.000 deg,	P =   0.000 deg,	R =   90.000 deg
};
P[2615]{
   GP1:
	UF : 0, UT : 6,		CONFIG : 'N U T, 0, 0, 0',
	X =  156.119  mm,	Y =   -231.540  mm,	Z =   -228.947  mm,
	W =  90.000 deg,	P =   0.000 deg,	R =   90.000 deg
};
P[2616]{
   GP1:
	UF : 0, UT : 6,		CONFIG : 'N U T, 0, 0, 0',
	X =  154.552  mm,	Y =   -232.574  mm,	Z =   -229.263  mm,
	W =  90.000 deg,	P =   0.000 deg,	R =   90.000 deg
};
P[2617]{
   GP1:
	UF : 0, UT : 6,		CONFIG : 'N U T, 0, 0, 0',
	X =  151.699  mm,	Y =   -234.190  mm,	Z =   -229.186  mm,
	W =  90.000 deg,	P =   0.000 deg,	R =   90.000 deg
};
P[2618]{
   GP1:
	UF : 0, UT : 6,		CONFIG : 'N U T, 0, 0, 0',
	X =  151.177  mm,	Y =   -234.545  mm,	Z =   -229.316  mm,
	W =  90.000 deg,	P =   0.000 deg,	R =   90.000 deg
};
P[2619]{
   GP1:
	UF : 0, UT : 6,		CONFIG : 'N U T, 0, 0, 0',
	X =  150.284  mm,	Y =   -235.042  mm,	Z =   -229.271  mm,
	W =  90.000 deg,	P =   0.000 deg,	R =   90.000 deg
};
P[2620]{
   GP1:
	UF : 0, UT : 6,		CONFIG : 'N U T, 0, 0, 0',
	X =  148.586  mm,	Y =   -235.940  mm,	Z =   -229.071  mm,
	W =  90.000 deg,	P =   0.000 deg,	R =   90.000 deg
};
P[2621]{
   GP1:
	UF : 0, UT : 6,		CONFIG : 'N U T, 0, 0, 0',
	X =  146.736  mm,	Y =   -236.986  mm,	Z =   -229.017  mm,
	W =  90.000 deg,	P =   0.000 deg,	R =   90.000 deg
};
P[2622]{
   GP1:
	UF : 0, UT : 6,		CONFIG : 'N U T, 0, 0, 0',
	X =  145.826  mm,	Y =   -237.471  mm,	Z =   -228.918  mm,
	W =  90.000 deg,	P =   0.000 deg,	R =   90.000 deg
};
P[2623]{
   GP1:
	UF : 0, UT : 6,		CONFIG : 'N U T, 0, 0, 0',
	X =  144.718  mm,	Y =   -238.173  mm,	Z =   -229.070  mm,
	W =  90.000 deg,	P =   0.000 deg,	R =   90.000 deg
};
P[2624]{
   GP1:
	UF : 0, UT : 6,		CONFIG : 'N U T, 0, 0, 0',
	X =  143.476  mm,	Y =   -239.008  mm,	Z =   -229.358  mm,
	W =  90.000 deg,	P =   0.000 deg,	R =   90.000 deg
};
P[2625]{
   GP1:
	UF : 0, UT : 6,		CONFIG : 'N U T, 0, 0, 0',
	X =  140.804  mm,	Y =   -240.446  mm,	Z =   -229.099  mm,
	W =  90.000 deg,	P =   0.000 deg,	R =   90.000 deg
};
P[2626]{
   GP1:
	UF : 0, UT : 6,		CONFIG : 'N U T, 0, 0, 0',
	X =  139.081  mm,	Y =   -241.439  mm,	Z =   -229.099  mm,
	W =  90.000 deg,	P =   0.000 deg,	R =   90.000 deg
};
P[2627]{
   GP1:
	UF : 0, UT : 6,		CONFIG : 'N U T, 0, 0, 0',
	X =  138.488  mm,	Y =   -241.830  mm,	Z =   -229.215  mm,
	W =  90.000 deg,	P =   0.000 deg,	R =   90.000 deg
};
P[2628]{
   GP1:
	UF : 0, UT : 6,		CONFIG : 'N U T, 0, 0, 0',
	X =  137.486  mm,	Y =   -242.303  mm,	Z =   -228.959  mm,
	W =  90.000 deg,	P =   0.000 deg,	R =   90.000 deg
};
P[2629]{
   GP1:
	UF : 0, UT : 6,		CONFIG : 'N U T, 0, 0, 0',
	X =  136.674  mm,	Y =   -242.894  mm,	Z =   -229.254  mm,
	W =  90.000 deg,	P =   0.000 deg,	R =   90.000 deg
};
P[2630]{
   GP1:
	UF : 0, UT : 6,		CONFIG : 'N U T, 0, 0, 0',
	X =  134.370  mm,	Y =   -244.187  mm,	Z =   -229.165  mm,
	W =  90.000 deg,	P =   0.000 deg,	R =   90.000 deg
};
P[2631]{
   GP1:
	UF : 0, UT : 6,		CONFIG : 'N U T, 0, 0, 0',
	X =  133.456  mm,	Y =   -244.622  mm,	Z =   -228.940  mm,
	W =  90.000 deg,	P =   0.000 deg,	R =   90.000 deg
};
P[2632]{
   GP1:
	UF : 0, UT : 6,		CONFIG : 'N U T, 0, 0, 0',
	X =  132.219  mm,	Y =   -245.480  mm,	Z =   -229.287  mm,
	W =  90.000 deg,	P =   0.000 deg,	R =   90.000 deg
};
P[2633]{
   GP1:
	UF : 0, UT : 6,		CONFIG : 'N U T, 0, 0, 0',
	X =  130.485  mm,	Y =   -246.355  mm,	Z =   -228.982  mm,
	W =  90.000 deg,	P =   0.000 deg,	R =   90.000 deg
};
P[2634]{
   GP1:
	UF : 0, UT : 6,		CONFIG : 'N U T, 0, 0, 0',
	X =  129.821  mm,	Y =   -246.824  mm,	Z =   -229.191  mm,
	W =  90.000 deg,	P =   0.000 deg,	R =   90.000 deg
};
P[2635]{
   GP1:
	UF : 0, UT : 6,		CONFIG : 'N U T, 0, 0, 0',
	X =  128.930  mm,	Y =   -247.226  mm,	Z =   -228.919  mm,
	W =  90.000 deg,	P =   0.000 deg,	R =   90.000 deg
};
P[2636]{
   GP1:
	UF : 0, UT : 6,		CONFIG : 'N U T, 0, 0, 0',
	X =  127.460  mm,	Y =   -248.171  mm,	Z =   -229.152  mm,
	W =  90.000 deg,	P =   0.000 deg,	R =   90.000 deg
};
P[2637]{
   GP1:
	UF : 0, UT : 6,		CONFIG : 'N U T, 0, 0, 0',
	X =  126.682  mm,	Y =   -248.579  mm,	Z =   -229.050  mm,
	W =  90.000 deg,	P =   0.000 deg,	R =   90.000 deg
};
P[2638]{
   GP1:
	UF : 0, UT : 6,		CONFIG : 'N U T, 0, 0, 0',
	X =  125.277  mm,	Y =   -249.467  mm,	Z =   -229.237  mm,
	W =  90.000 deg,	P =   0.000 deg,	R =   90.000 deg
};
P[2639]{
   GP1:
	UF : 0, UT : 6,		CONFIG : 'N U T, 0, 0, 0',
	X =  124.553  mm,	Y =   -249.822  mm,	Z =   -229.086  mm,
	W =  90.000 deg,	P =   0.000 deg,	R =   90.000 deg
};
P[2640]{
   GP1:
	UF : 0, UT : 6,		CONFIG : 'N U T, 0, 0, 0',
	X =  122.567  mm,	Y =   -250.988  mm,	Z =   -229.132  mm,
	W =  90.000 deg,	P =   0.000 deg,	R =   90.000 deg
};
P[2641]{
   GP1:
	UF : 0, UT : 6,		CONFIG : 'N U T, 0, 0, 0',
	X =  121.584  mm,	Y =   -251.623  mm,	Z =   -229.295  mm,
	W =  90.000 deg,	P =   0.000 deg,	R =   90.000 deg
};
P[2642]{
   GP1:
	UF : 0, UT : 6,		CONFIG : 'N U T, 0, 0, 0',
	X =  120.813  mm,	Y =   -252.077  mm,	Z =   -229.316  mm,
	W =  90.000 deg,	P =   0.000 deg,	R =   90.000 deg
};
P[2643]{
   GP1:
	UF : 0, UT : 6,		CONFIG : 'N U T, 0, 0, 0',
	X =  119.548  mm,	Y =   -252.647  mm,	Z =   -228.925  mm,
	W =  90.000 deg,	P =   0.000 deg,	R =   90.000 deg
};
P[2644]{
   GP1:
	UF : 0, UT : 6,		CONFIG : 'N U T, 0, 0, 0',
	X =  115.743  mm,	Y =   -254.946  mm,	Z =   -229.174  mm,
	W =  90.000 deg,	P =   0.000 deg,	R =   90.000 deg
};
P[2645]{
   GP1:
	UF : 0, UT : 6,		CONFIG : 'N U T, 0, 0, 0',
	X =  114.979  mm,	Y =   -255.410  mm,	Z =   -229.232  mm,
	W =  90.000 deg,	P =   0.000 deg,	R =   90.000 deg
};
P[2646]{
   GP1:
	UF : 0, UT : 6,		CONFIG : 'N U T, 0, 0, 0',
	X =  113.976  mm,	Y =   -255.972  mm,	Z =   -229.188  mm,
	W =  90.000 deg,	P =   0.000 deg,	R =   90.000 deg
};
P[2647]{
   GP1:
	UF : 0, UT : 6,		CONFIG : 'N U T, 0, 0, 0',
	X =  111.329  mm,	Y =   -257.525  mm,	Z =   -229.249  mm,
	W =  90.000 deg,	P =   0.000 deg,	R =   90.000 deg
};
P[2648]{
   GP1:
	UF : 0, UT : 6,		CONFIG : 'N U T, 0, 0, 0',
	X =  110.284  mm,	Y =   -258.152  mm,	Z =   -229.306  mm,
	W =  90.000 deg,	P =   0.000 deg,	R =   90.000 deg
};
P[2649]{
   GP1:
	UF : 0, UT : 6,		CONFIG : 'N U T, 0, 0, 0',
	X =  109.545  mm,	Y =   -258.446  mm,	Z =   -228.985  mm,
	W =  90.000 deg,	P =   0.000 deg,	R =   90.000 deg
};
P[2650]{
   GP1:
	UF : 0, UT : 6,		CONFIG : 'N U T, 0, 0, 0',
	X =  108.379  mm,	Y =   -259.147  mm,	Z =   -229.051  mm,
	W =  90.000 deg,	P =   0.000 deg,	R =   90.000 deg
};
P[2651]{
   GP1:
	UF : 0, UT : 6,		CONFIG : 'N U T, 0, 0, 0',
	X =  195.000  mm,	Y =   -410.000  mm,	Z =   -170.000  mm,
	W =  90.000 deg,	P =   0.000 deg,	R =   90.000 deg
};
/END
